(* CODESYS project TASK3.project
   CompiledLibraryCompatibilityVersion: LeadSysStudio V3.5 SP15 Patch 4
   Title: TASK3

Project tree, tasks and I/O mapping:
  Device : PMC600, Leadshine Technology Co., Ltd., order no. 600101, version 3.5.15.40
    application Application
      libraries: Standard, * (System)
      task MainTask (cyclic, interval t#4ms, priority 4, watchdog t#5000ms x 1) calls nothing
      task EtherCAT_Master_Leadshine_A (cyclic, interval 4000 µs, priority 0) calls PLC_PRG, EtherCAT_Master_Leadshine_A.EtherCAT_Task
      task SoftMotion_PlanningTask (freewheeling, priority 15) calls nothing
      program PLC_PRG [LD]
      axis group Tripod: TRAFO.Kin_Tripod_Rotary, axes Axis_3, Axis_4, Axis_5
    Device Diagnose
    Network Configuration
      LocalBus Config
    Resource Usage
    SoftMotion General Axis Pool
    High_Speed_IO_Module : High Speed IO Module, Leadshine Technology Co., Ltd., version 3.5.15.40
        unmapped channels: Genral_IO_IN, Genral_IO_Out
    EtherCAT_Master_Leadshine_A : EtherCAT Master Leadshine, Leadshine Technology Co., Ltd., version 3.5.9.50
        settings: MasterCycleTime = 4000
      PM32EC_LOCAL : PM32EC-LOCAL, Leadshine Technology Co., Ltd., order no. PM32EC-LOCAL, version Revision=16#20061010
          settings: StationAlias = 0; DC sync0 cycletime = 4000; DC sync1 cycletime = 4000
      DM3C_EC522 : DM3C-EC522(COE), Leadshine Technology Co.,Ltd., order no. DM3C-EC522, version Revision=16#00000001
          settings: StationAlias = 0; DC sync0 cycletime = 4000; DC sync1 cycletime = 4000; Number of SDO = 6; Homing method.Index = 16#6098; Homing method.Subindex = 16#00; Homing method.Value = 29; Homing method.Size = 8; Homing method.AbortIfError = FALSE; Homing method.JumpToLine = FALSE; Homing method.Line = 0; Homing method.CompleteAccess = FALSE; Homing velocity (fast).Index = 16#6099; Homing velocity (fast).Subindex = 16#01; Homing velocity (fast).Value = 1667; Homing velocity (fast).Size = 32; Homing velocity (fast).AbortIfError = FALSE; Homing velocity (fast).JumpToLine = FALSE; Homing velocity (fast).Line = 0; Homing velocity (fast).CompleteAccess = FALSE; Homing velocity (slow).Index = 16#6099; Homing velocity (slow).Subindex = 16#02; Homing velocity (slow).Value = 333; Homing velocity (slow).Size = 32; Homing velocity (slow).AbortIfError = FALSE; Homing velocity (slow).JumpToLine = FALSE; Homing velocity (slow).Line = 0; Homing velocity (slow).CompleteAccess = FALSE; Homing acceleration.Index = 16#609A; Homing acceleration.Subindex = 16#00; Homing acceleration.Value = 16667; Homing acceleration.Size = 32; Homing acceleration.AbortIfError = FALSE; Homing acceleration.JumpToLine = FALSE; Homing acceleration.Line = 0; Homing acceleration.CompleteAccess = FALSE; Homing offset.Index = 16#607C; Homing offset.Subindex = 16#00; Homing offset.Value = 0; Homing offset.Size = 32;
            Homing offset.AbortIfError = FALSE; Homing offset.JumpToLine = FALSE; Homing offset.Line = 0; Homing offset.CompleteAccess = FALSE
          unmapped channels: Control Word, Profile Target Position, Touch Probe Function, Last Error Code, Status Word, Modes of Operation display, Position Actual Value, Touch Probe Status, Touch Probe 1 Positive Value, Digital Inputs
        Axis : Axis, 3S - Smart Software Solutions GmbH, order no. 0, version 4.6.1.0
            settings: wDriveID = 0; dwRatioTechUnitsDenom = 500; iRatioTechUnitsNum = 3; 一圈脉冲数 = 10000; 工作台一圈的位移 = 60; 电子齿轮比分子 = 1; 电子齿轮比分母 = 1; ScalingIncs = 500; ScalingUnits = 3; AdrOffset_8010 = 4; BitOffset_8010 = 0; BitLength_8010 = 16; Address_8010 = '%QW2'; Type_8010 = 'UINT'; AddressPointer_8010 = ADR(%QW2); AdrOffset_8020 = 8; BitOffset_8020 = 0; BitLength_8020 = 32; Address_8020 = '%QD2'; Type_8020 = 'DINT'; AddressPointer_8020 = ADR(%QD2); AdrOffset_8030 = 4294967295; BitOffset_8030 = 0; BitLength_8030 = 32; Address_8030 = ''; Type_8030 = 'DINT'; AddressPointer_8030 = 0; AdrOffset_8040 = 4294967295; BitOffset_8040 = 0; BitLength_8040 = 0; Address_8040 = ''; Type_8040 = ''; AddressPointer_8040 = 0; AdrOffset_8050 = 4294967295; BitOffset_8050 = 0; BitLength_8050 = 8; Address_8050 = ''; Type_8050 = 'USINT'; AddressPointer_8050 = 0; AdrOffset_8060 = 12;
              BitOffset_8060 = 0; BitLength_8060 = 16; Address_8060 = '%QW6'; Type_8060 = 'UINT'; AddressPointer_8060 = ADR(%QW6); AdrOffset_8070 = 4294967295; BitOffset_8070 = 0; BitLength_8070 = 0; Address_8070 = ''; Type_8070 = ''; AddressPointer_8070 = 0; AdrOffset_8080 = 4294967295; BitOffset_8080 = 0; BitLength_8080 = 0; Address_8080 = ''; Type_8080 = ''; AddressPointer_8080 = 0; AdrOffset_8090 = 4294967295; BitOffset_8090 = 0; BitLength_8090 = 0; Address_8090 = ''; Type_8090 = ''; AddressPointer_8090 = 0; AdrOffset_8510 = 6; BitOffset_8510 = 0; BitLength_8510 = 16; Address_8510 = '%IW3'; Type_8510 = 'UINT'; AddressPointer_8510 = ADR(%IW3); AdrOffset_8520 = 12; BitOffset_8520 = 0; BitLength_8520 = 32; Address_8520 = '%ID3'; Type_8520 = 'DINT'; AddressPointer_8520 = ADR(%ID3); AdrOffset_8530 = 4294967295; BitOffset_8530 = 0; BitLength_8530 = 0; Address_8530 = ''; Type_8530 = '';
              AddressPointer_8530 = 0; AdrOffset_8540 = 4294967295; BitOffset_8540 = 0; BitLength_8540 = 0; Address_8540 = ''; Type_8540 = ''; AddressPointer_8540 = 0; AdrOffset_8550 = 8; BitOffset_8550 = 0; BitLength_8550 = 8; Address_8550 = '%IB8'; Type_8550 = 'SINT'; AddressPointer_8550 = ADR(%IB8); AdrOffset_8560 = 24; BitOffset_8560 = 0; BitLength_8560 = 32; Address_8560 = '%ID6'; Type_8560 = 'UDINT'; AddressPointer_8560 = ADR(%ID6); AdrOffset_8570 = 16; BitOffset_8570 = 0; BitLength_8570 = 16; Address_8570 = '%IW8'; Type_8570 = 'UINT'; AddressPointer_8570 = ADR(%IW8); AdrOffset_8580 = 20; BitOffset_8580 = 0; BitLength_8580 = 32; Address_8580 = '%ID5'; Type_8580 = 'DINT'; AddressPointer_8580 = ADR(%ID5); AdrOffset_8590 = 4294967295; BitOffset_8590 = 0; BitLength_8590 = 0; Address_8590 = ''; Type_8590 = ''; AddressPointer_8590 = 0; AdrOffset_8600 = 4294967295; BitOffset_8600 = 0; BitLength_8600 = 0;
              Address_8600 = ''; Type_8600 = ''; AddressPointer_8600 = 0; AdrOffset_8600 = 4294967295; BitOffset_8600 = 0; BitLength_8600 = 0; Address_8610 = ''; Type_8610 = ''; AddressPointer_8610 = 0; AdrOffset_8620 = 4294967295; BitOffset_8620 = 0; BitLength_8620 = 0; Address_8620 = ''; Type_8620 = ''; AddressPointer_8620 = 0
      DM3C_EC522_1 : DM3C-EC522(COE), Leadshine Technology Co.,Ltd., order no. DM3C-EC522, version Revision=16#00000001
          settings: StationAlias = 0; DC sync0 cycletime = 4000; DC sync1 cycletime = 4000; Number of SDO = 6; Homing method.Index = 16#6098; Homing method.Subindex = 16#00; Homing method.Value = 29; Homing method.Size = 8; Homing method.AbortIfError = FALSE; Homing method.JumpToLine = FALSE; Homing method.Line = 0; Homing method.CompleteAccess = FALSE; Homing velocity (fast).Index = 16#6099; Homing velocity (fast).Subindex = 16#01; Homing velocity (fast).Value = 1667; Homing velocity (fast).Size = 32; Homing velocity (fast).AbortIfError = FALSE; Homing velocity (fast).JumpToLine = FALSE; Homing velocity (fast).Line = 0; Homing velocity (fast).CompleteAccess = FALSE; Homing velocity (slow).Index = 16#6099; Homing velocity (slow).Subindex = 16#02; Homing velocity (slow).Value = 333; Homing velocity (slow).Size = 32; Homing velocity (slow).AbortIfError = FALSE; Homing velocity (slow).JumpToLine = FALSE; Homing velocity (slow).Line = 0; Homing velocity (slow).CompleteAccess = FALSE; Homing acceleration.Index = 16#609A; Homing acceleration.Subindex = 16#00; Homing acceleration.Value = 16667; Homing acceleration.Size = 32; Homing acceleration.AbortIfError = FALSE; Homing acceleration.JumpToLine = FALSE; Homing acceleration.Line = 0; Homing acceleration.CompleteAccess = FALSE; Homing offset.Index = 16#607C; Homing offset.Subindex = 16#00; Homing offset.Value = 0; Homing offset.Size = 32;
            Homing offset.AbortIfError = FALSE; Homing offset.JumpToLine = FALSE; Homing offset.Line = 0; Homing offset.CompleteAccess = FALSE
          unmapped channels: Control Word, Profile Target Position, Touch Probe Function, Last Error Code, Status Word, Modes of Operation display, Position Actual Value, Touch Probe Status, Touch Probe 1 Positive Value, Digital Inputs
        Axis_1 : Axis, 3S - Smart Software Solutions GmbH, order no. 0, version 4.6.1.0
            settings: dwRatioTechUnitsDenom = 500; iRatioTechUnitsNum = 3; 一圈脉冲数 = 10000; 工作台一圈的位移 = 60; 电子齿轮比分子 = 1; 电子齿轮比分母 = 1; ScalingIncs = 500; ScalingUnits = 3; AdrOffset_8010 = 16; BitOffset_8010 = 0; BitLength_8010 = 16; Address_8010 = '%QW8'; Type_8010 = 'UINT'; AddressPointer_8010 = ADR(%QW8); AdrOffset_8020 = 20; BitOffset_8020 = 0; BitLength_8020 = 32; Address_8020 = '%QD5'; Type_8020 = 'DINT'; AddressPointer_8020 = ADR(%QD5); AdrOffset_8030 = 4294967295; BitOffset_8030 = 0; BitLength_8030 = 32; Address_8030 = ''; Type_8030 = 'DINT'; AddressPointer_8030 = 0; AdrOffset_8040 = 4294967295; BitOffset_8040 = 0; BitLength_8040 = 0; Address_8040 = ''; Type_8040 = ''; AddressPointer_8040 = 0; AdrOffset_8050 = 4294967295; BitOffset_8050 = 0; BitLength_8050 = 8; Address_8050 = ''; Type_8050 = 'USINT'; AddressPointer_8050 = 0; AdrOffset_8060 = 24; BitOffset_8060 = 0;
              BitLength_8060 = 16; Address_8060 = '%QW12'; Type_8060 = 'UINT'; AddressPointer_8060 = ADR(%QW12); AdrOffset_8070 = 4294967295; BitOffset_8070 = 0; BitLength_8070 = 0; Address_8070 = ''; Type_8070 = ''; AddressPointer_8070 = 0; AdrOffset_8080 = 4294967295; BitOffset_8080 = 0; BitLength_8080 = 0; Address_8080 = ''; Type_8080 = ''; AddressPointer_8080 = 0; AdrOffset_8090 = 4294967295; BitOffset_8090 = 0; BitLength_8090 = 0; Address_8090 = ''; Type_8090 = ''; AddressPointer_8090 = 0; AdrOffset_8510 = 30; BitOffset_8510 = 0; BitLength_8510 = 16; Address_8510 = '%IW15'; Type_8510 = 'UINT'; AddressPointer_8510 = ADR(%IW15); AdrOffset_8520 = 36; BitOffset_8520 = 0; BitLength_8520 = 32; Address_8520 = '%ID9'; Type_8520 = 'DINT'; AddressPointer_8520 = ADR(%ID9); AdrOffset_8530 = 4294967295; BitOffset_8530 = 0; BitLength_8530 = 0; Address_8530 = ''; Type_8530 = ''; AddressPointer_8530 = 0;
              AdrOffset_8540 = 4294967295; BitOffset_8540 = 0; BitLength_8540 = 0; Address_8540 = ''; Type_8540 = ''; AddressPointer_8540 = 0; AdrOffset_8550 = 32; BitOffset_8550 = 0; BitLength_8550 = 8; Address_8550 = '%IB32'; Type_8550 = 'SINT'; AddressPointer_8550 = ADR(%IB32); AdrOffset_8560 = 48; BitOffset_8560 = 0; BitLength_8560 = 32; Address_8560 = '%ID12'; Type_8560 = 'UDINT'; AddressPointer_8560 = ADR(%ID12); AdrOffset_8570 = 40; BitOffset_8570 = 0; BitLength_8570 = 16; Address_8570 = '%IW20'; Type_8570 = 'UINT'; AddressPointer_8570 = ADR(%IW20); AdrOffset_8580 = 44; BitOffset_8580 = 0; BitLength_8580 = 32; Address_8580 = '%ID11'; Type_8580 = 'DINT'; AddressPointer_8580 = ADR(%ID11); AdrOffset_8590 = 4294967295; BitOffset_8590 = 0; BitLength_8590 = 0; Address_8590 = ''; Type_8590 = ''; AddressPointer_8590 = 0; AdrOffset_8600 = 4294967295; BitOffset_8600 = 0; BitLength_8600 = 0; Address_8600 = '';
              Type_8600 = ''; AddressPointer_8600 = 0; AdrOffset_8600 = 4294967295; BitOffset_8600 = 0; BitLength_8600 = 0; Address_8610 = ''; Type_8610 = ''; AddressPointer_8610 = 0; AdrOffset_8620 = 4294967295; BitOffset_8620 = 0; BitLength_8620 = 0; Address_8620 = ''; Type_8620 = ''; AddressPointer_8620 = 0
      DM3C_EC522_2 : DM3C-EC522(COE), Leadshine Technology Co.,Ltd., order no. DM3C-EC522, version Revision=16#00000001
          settings: StationAlias = 0; DC sync0 cycletime = 4000; DC sync1 cycletime = 4000; Number of SDO = 6; Homing method.Index = 16#6098; Homing method.Subindex = 16#00; Homing method.Value = 29; Homing method.Size = 8; Homing method.AbortIfError = FALSE; Homing method.JumpToLine = FALSE; Homing method.Line = 0; Homing method.CompleteAccess = FALSE; Homing velocity (fast).Index = 16#6099; Homing velocity (fast).Subindex = 16#01; Homing velocity (fast).Value = 25000; Homing velocity (fast).Size = 32; Homing velocity (fast).AbortIfError = FALSE; Homing velocity (fast).JumpToLine = FALSE; Homing velocity (fast).Line = 0; Homing velocity (fast).CompleteAccess = FALSE; Homing velocity (slow).Index = 16#6099; Homing velocity (slow).Subindex = 16#02; Homing velocity (slow).Value = 5000; Homing velocity (slow).Size = 32; Homing velocity (slow).AbortIfError = FALSE; Homing velocity (slow).JumpToLine = FALSE; Homing velocity (slow).Line = 0; Homing velocity (slow).CompleteAccess = FALSE; Homing acceleration.Index = 16#609A; Homing acceleration.Subindex = 16#00; Homing acceleration.Value = 250000; Homing acceleration.Size = 32; Homing acceleration.AbortIfError = FALSE; Homing acceleration.JumpToLine = FALSE; Homing acceleration.Line = 0; Homing acceleration.CompleteAccess = FALSE; Homing offset.Index = 16#607C; Homing offset.Subindex = 16#00; Homing offset.Value = 0; Homing offset.Size = 32;
            Homing offset.AbortIfError = FALSE; Homing offset.JumpToLine = FALSE; Homing offset.Line = 0; Homing offset.CompleteAccess = FALSE
          unmapped channels: Control Word, Profile Target Position, Touch Probe Function, Last Error Code, Status Word, Modes of Operation display, Position Actual Value, Touch Probe Status, Touch Probe 1 Positive Value, Digital Inputs
        Axis_2 : Axis, 3S - Smart Software Solutions GmbH, order no. 0, version 4.6.1.0
            settings: wDriveID = 2; dwRatioTechUnitsDenom = 2500; 一圈脉冲数 = 10000; 工作台一圈的位移 = 4; 电子齿轮比分子 = 1; 电子齿轮比分母 = 1; ScalingIncs = 2500; AdrOffset_8010 = 28; BitOffset_8010 = 0; BitLength_8010 = 16; Address_8010 = '%QW14'; Type_8010 = 'UINT'; AddressPointer_8010 = ADR(%QW14); AdrOffset_8020 = 32; BitOffset_8020 = 0; BitLength_8020 = 32; Address_8020 = '%QD8'; Type_8020 = 'DINT'; AddressPointer_8020 = ADR(%QD8); AdrOffset_8030 = 4294967295; BitOffset_8030 = 0; BitLength_8030 = 32; Address_8030 = ''; Type_8030 = 'DINT'; AddressPointer_8030 = 0; AdrOffset_8040 = 4294967295; BitOffset_8040 = 0; BitLength_8040 = 0; Address_8040 = ''; Type_8040 = ''; AddressPointer_8040 = 0; AdrOffset_8050 = 4294967295; BitOffset_8050 = 0; BitLength_8050 = 8; Address_8050 = ''; Type_8050 = 'USINT'; AddressPointer_8050 = 0; AdrOffset_8060 = 36; BitOffset_8060 = 0; BitLength_8060 = 16;
              Address_8060 = '%QW18'; Type_8060 = 'UINT'; AddressPointer_8060 = ADR(%QW18); AdrOffset_8070 = 4294967295; BitOffset_8070 = 0; BitLength_8070 = 0; Address_8070 = ''; Type_8070 = ''; AddressPointer_8070 = 0; AdrOffset_8080 = 4294967295; BitOffset_8080 = 0; BitLength_8080 = 0; Address_8080 = ''; Type_8080 = ''; AddressPointer_8080 = 0; AdrOffset_8090 = 4294967295; BitOffset_8090 = 0; BitLength_8090 = 0; Address_8090 = ''; Type_8090 = ''; AddressPointer_8090 = 0; AdrOffset_8510 = 54; BitOffset_8510 = 0; BitLength_8510 = 16; Address_8510 = '%IW27'; Type_8510 = 'UINT'; AddressPointer_8510 = ADR(%IW27); AdrOffset_8520 = 60; BitOffset_8520 = 0; BitLength_8520 = 32; Address_8520 = '%ID15'; Type_8520 = 'DINT'; AddressPointer_8520 = ADR(%ID15); AdrOffset_8530 = 4294967295; BitOffset_8530 = 0; BitLength_8530 = 0; Address_8530 = ''; Type_8530 = ''; AddressPointer_8530 = 0; AdrOffset_8540 = 4294967295;
              BitOffset_8540 = 0; BitLength_8540 = 0; Address_8540 = ''; Type_8540 = ''; AddressPointer_8540 = 0; AdrOffset_8550 = 56; BitOffset_8550 = 0; BitLength_8550 = 8; Address_8550 = '%IB56'; Type_8550 = 'SINT'; AddressPointer_8550 = ADR(%IB56); AdrOffset_8560 = 72; BitOffset_8560 = 0; BitLength_8560 = 32; Address_8560 = '%ID18'; Type_8560 = 'UDINT'; AddressPointer_8560 = ADR(%ID18); AdrOffset_8570 = 64; BitOffset_8570 = 0; BitLength_8570 = 16; Address_8570 = '%IW32'; Type_8570 = 'UINT'; AddressPointer_8570 = ADR(%IW32); AdrOffset_8580 = 68; BitOffset_8580 = 0; BitLength_8580 = 32; Address_8580 = '%ID17'; Type_8580 = 'DINT'; AddressPointer_8580 = ADR(%ID17); AdrOffset_8590 = 4294967295; BitOffset_8590 = 0; BitLength_8590 = 0; Address_8590 = ''; Type_8590 = ''; AddressPointer_8590 = 0; AdrOffset_8600 = 4294967295; BitOffset_8600 = 0; BitLength_8600 = 0; Address_8600 = ''; Type_8600 = '';
              AddressPointer_8600 = 0; AdrOffset_8600 = 4294967295; BitOffset_8600 = 0; BitLength_8600 = 0; Address_8610 = ''; Type_8610 = ''; AddressPointer_8610 = 0; AdrOffset_8620 = 4294967295; BitOffset_8620 = 0; BitLength_8620 = 0; Address_8620 = ''; Type_8620 = ''; AddressPointer_8620 = 0
      DM3C_EC522_3 : DM3C-EC522(COE), Leadshine Technology Co.,Ltd., order no. DM3C-EC522, version Revision=16#00000001
          settings: StationAlias = 0; DC sync0 cycletime = 4000; DC sync1 cycletime = 4000; Number of SDO = 6; Homing method.Index = 16#6098; Homing method.Subindex = 16#00; Homing method.Value = 21; Homing method.Size = 8; Homing method.AbortIfError = FALSE; Homing method.JumpToLine = FALSE; Homing method.Line = 0; Homing method.CompleteAccess = FALSE; Homing velocity (fast).Index = 16#6099; Homing velocity (fast).Subindex = 16#01; Homing velocity (fast).Value = 7500; Homing velocity (fast).Size = 32; Homing velocity (fast).AbortIfError = FALSE; Homing velocity (fast).JumpToLine = FALSE; Homing velocity (fast).Line = 0; Homing velocity (fast).CompleteAccess = FALSE; Homing velocity (slow).Index = 16#6099; Homing velocity (slow).Subindex = 16#02; Homing velocity (slow).Value = 5000; Homing velocity (slow).Size = 32; Homing velocity (slow).AbortIfError = FALSE; Homing velocity (slow).JumpToLine = FALSE; Homing velocity (slow).Line = 0; Homing velocity (slow).CompleteAccess = FALSE; Homing acceleration.Index = 16#609A; Homing acceleration.Subindex = 16#00; Homing acceleration.Value = 50000; Homing acceleration.Size = 32; Homing acceleration.AbortIfError = FALSE; Homing acceleration.JumpToLine = FALSE; Homing acceleration.Line = 0; Homing acceleration.CompleteAccess = FALSE; Homing offset.Index = 16#607C; Homing offset.Subindex = 16#00; Homing offset.Value = 0; Homing offset.Size = 32;
            Homing offset.AbortIfError = FALSE; Homing offset.JumpToLine = FALSE; Homing offset.Line = 0; Homing offset.CompleteAccess = FALSE
          unmapped channels: Control Word, Profile Target Position, Touch Probe Function, Last Error Code, Status Word, Modes of Operation display, Position Actual Value, Touch Probe Status, Touch Probe 1 Positive Value, Digital Inputs
        Axis_3 : Axis, 3S - Smart Software Solutions GmbH, order no. 0, version 4.6.1.0
            settings: wDriveID = 3; dwRatioTechUnitsDenom = 500; iRatioTechUnitsNum = -1; 一圈脉冲数 = 36000; 工作台一圈的位移 = 360; 电子齿轮比分子 = 5; 电子齿轮比分母 = 1; ScalingIncs = 500; InvertDirection = True; AdrOffset_8010 = 40; BitOffset_8010 = 0; BitLength_8010 = 16; Address_8010 = '%QW20'; Type_8010 = 'UINT'; AddressPointer_8010 = ADR(%QW20); AdrOffset_8020 = 44; BitOffset_8020 = 0; BitLength_8020 = 32; Address_8020 = '%QD11'; Type_8020 = 'DINT'; AddressPointer_8020 = ADR(%QD11); AdrOffset_8030 = 4294967295; BitOffset_8030 = 0; BitLength_8030 = 32; Address_8030 = ''; Type_8030 = 'DINT'; AddressPointer_8030 = 0; AdrOffset_8040 = 4294967295; BitOffset_8040 = 0; BitLength_8040 = 0; Address_8040 = ''; Type_8040 = ''; AddressPointer_8040 = 0; AdrOffset_8050 = 4294967295; BitOffset_8050 = 0; BitLength_8050 = 8; Address_8050 = ''; Type_8050 = 'USINT'; AddressPointer_8050 = 0; AdrOffset_8060 = 48;
              BitOffset_8060 = 0; BitLength_8060 = 16; Address_8060 = '%QW24'; Type_8060 = 'UINT'; AddressPointer_8060 = ADR(%QW24); AdrOffset_8070 = 4294967295; BitOffset_8070 = 0; BitLength_8070 = 0; Address_8070 = ''; Type_8070 = ''; AddressPointer_8070 = 0; AdrOffset_8080 = 4294967295; BitOffset_8080 = 0; BitLength_8080 = 0; Address_8080 = ''; Type_8080 = ''; AddressPointer_8080 = 0; AdrOffset_8090 = 4294967295; BitOffset_8090 = 0; BitLength_8090 = 0; Address_8090 = ''; Type_8090 = ''; AddressPointer_8090 = 0; AdrOffset_8510 = 78; BitOffset_8510 = 0; BitLength_8510 = 16; Address_8510 = '%IW39'; Type_8510 = 'UINT'; AddressPointer_8510 = ADR(%IW39); AdrOffset_8520 = 84; BitOffset_8520 = 0; BitLength_8520 = 32; Address_8520 = '%ID21'; Type_8520 = 'DINT'; AddressPointer_8520 = ADR(%ID21); AdrOffset_8530 = 4294967295; BitOffset_8530 = 0; BitLength_8530 = 0; Address_8530 = ''; Type_8530 = '';
              AddressPointer_8530 = 0; AdrOffset_8540 = 4294967295; BitOffset_8540 = 0; BitLength_8540 = 0; Address_8540 = ''; Type_8540 = ''; AddressPointer_8540 = 0; AdrOffset_8550 = 80; BitOffset_8550 = 0; BitLength_8550 = 8; Address_8550 = '%IB80'; Type_8550 = 'SINT'; AddressPointer_8550 = ADR(%IB80); AdrOffset_8560 = 96; BitOffset_8560 = 0; BitLength_8560 = 32; Address_8560 = '%ID24'; Type_8560 = 'UDINT'; AddressPointer_8560 = ADR(%ID24); AdrOffset_8570 = 88; BitOffset_8570 = 0; BitLength_8570 = 16; Address_8570 = '%IW44'; Type_8570 = 'UINT'; AddressPointer_8570 = ADR(%IW44); AdrOffset_8580 = 92; BitOffset_8580 = 0; BitLength_8580 = 32; Address_8580 = '%ID23'; Type_8580 = 'DINT'; AddressPointer_8580 = ADR(%ID23); AdrOffset_8590 = 4294967295; BitOffset_8590 = 0; BitLength_8590 = 0; Address_8590 = ''; Type_8590 = ''; AddressPointer_8590 = 0; AdrOffset_8600 = 4294967295; BitOffset_8600 = 0; BitLength_8600 = 0;
              Address_8600 = ''; Type_8600 = ''; AddressPointer_8600 = 0; AdrOffset_8600 = 4294967295; BitOffset_8600 = 0; BitLength_8600 = 0; Address_8610 = ''; Type_8610 = ''; AddressPointer_8610 = 0; AdrOffset_8620 = 4294967295; BitOffset_8620 = 0; BitLength_8620 = 0; Address_8620 = ''; Type_8620 = ''; AddressPointer_8620 = 0
      DM3C_EC522_4 : DM3C-EC522(COE), Leadshine Technology Co.,Ltd., order no. DM3C-EC522, version Revision=16#00000001
          settings: StationAlias = 0; DC sync0 cycletime = 4000; DC sync1 cycletime = 4000; Number of SDO = 6; Homing method.Index = 16#6098; Homing method.Subindex = 16#00; Homing method.Value = 21; Homing method.Size = 8; Homing method.AbortIfError = FALSE; Homing method.JumpToLine = FALSE; Homing method.Line = 0; Homing method.CompleteAccess = FALSE; Homing velocity (fast).Index = 16#6099; Homing velocity (fast).Subindex = 16#01; Homing velocity (fast).Value = 7500; Homing velocity (fast).Size = 32; Homing velocity (fast).AbortIfError = FALSE; Homing velocity (fast).JumpToLine = FALSE; Homing velocity (fast).Line = 0; Homing velocity (fast).CompleteAccess = FALSE; Homing velocity (slow).Index = 16#6099; Homing velocity (slow).Subindex = 16#02; Homing velocity (slow).Value = 5000; Homing velocity (slow).Size = 32; Homing velocity (slow).AbortIfError = FALSE; Homing velocity (slow).JumpToLine = FALSE; Homing velocity (slow).Line = 0; Homing velocity (slow).CompleteAccess = FALSE; Homing acceleration.Index = 16#609A; Homing acceleration.Subindex = 16#00; Homing acceleration.Value = 50000; Homing acceleration.Size = 32; Homing acceleration.AbortIfError = FALSE; Homing acceleration.JumpToLine = FALSE; Homing acceleration.Line = 0; Homing acceleration.CompleteAccess = FALSE; Homing offset.Index = 16#607C; Homing offset.Subindex = 16#00; Homing offset.Value = 0; Homing offset.Size = 32;
            Homing offset.AbortIfError = FALSE; Homing offset.JumpToLine = FALSE; Homing offset.Line = 0; Homing offset.CompleteAccess = FALSE
          unmapped channels: Control Word, Profile Target Position, Touch Probe Function, Last Error Code, Status Word, Modes of Operation display, Position Actual Value, Touch Probe Status, Touch Probe 1 Positive Value, Digital Inputs
        Axis_4 : Axis, 3S - Smart Software Solutions GmbH, order no. 0, version 4.6.1.0
            settings: wDriveID = 4; dwRatioTechUnitsDenom = 500; iRatioTechUnitsNum = -1; 一圈脉冲数 = 36000; 工作台一圈的位移 = 360; 电子齿轮比分子 = 5; 电子齿轮比分母 = 1; ScalingIncs = 500; InvertDirection = True; AdrOffset_8010 = 52; BitOffset_8010 = 0; BitLength_8010 = 16; Address_8010 = '%QW26'; Type_8010 = 'UINT'; AddressPointer_8010 = ADR(%QW26); AdrOffset_8020 = 56; BitOffset_8020 = 0; BitLength_8020 = 32; Address_8020 = '%QD14'; Type_8020 = 'DINT'; AddressPointer_8020 = ADR(%QD14); AdrOffset_8030 = 4294967295; BitOffset_8030 = 0; BitLength_8030 = 32; Address_8030 = ''; Type_8030 = 'DINT'; AddressPointer_8030 = 0; AdrOffset_8040 = 4294967295; BitOffset_8040 = 0; BitLength_8040 = 0; Address_8040 = ''; Type_8040 = ''; AddressPointer_8040 = 0; AdrOffset_8050 = 4294967295; BitOffset_8050 = 0; BitLength_8050 = 8; Address_8050 = ''; Type_8050 = 'USINT'; AddressPointer_8050 = 0; AdrOffset_8060 = 60;
              BitOffset_8060 = 0; BitLength_8060 = 16; Address_8060 = '%QW30'; Type_8060 = 'UINT'; AddressPointer_8060 = ADR(%QW30); AdrOffset_8070 = 4294967295; BitOffset_8070 = 0; BitLength_8070 = 0; Address_8070 = ''; Type_8070 = ''; AddressPointer_8070 = 0; AdrOffset_8080 = 4294967295; BitOffset_8080 = 0; BitLength_8080 = 0; Address_8080 = ''; Type_8080 = ''; AddressPointer_8080 = 0; AdrOffset_8090 = 4294967295; BitOffset_8090 = 0; BitLength_8090 = 0; Address_8090 = ''; Type_8090 = ''; AddressPointer_8090 = 0; AdrOffset_8510 = 102; BitOffset_8510 = 0; BitLength_8510 = 16; Address_8510 = '%IW51'; Type_8510 = 'UINT'; AddressPointer_8510 = ADR(%IW51); AdrOffset_8520 = 108; BitOffset_8520 = 0; BitLength_8520 = 32; Address_8520 = '%ID27'; Type_8520 = 'DINT'; AddressPointer_8520 = ADR(%ID27); AdrOffset_8530 = 4294967295; BitOffset_8530 = 0; BitLength_8530 = 0; Address_8530 = ''; Type_8530 = '';
              AddressPointer_8530 = 0; AdrOffset_8540 = 4294967295; BitOffset_8540 = 0; BitLength_8540 = 0; Address_8540 = ''; Type_8540 = ''; AddressPointer_8540 = 0; AdrOffset_8550 = 104; BitOffset_8550 = 0; BitLength_8550 = 8; Address_8550 = '%IB104'; Type_8550 = 'SINT'; AddressPointer_8550 = ADR(%IB104); AdrOffset_8560 = 120; BitOffset_8560 = 0; BitLength_8560 = 32; Address_8560 = '%ID30'; Type_8560 = 'UDINT'; AddressPointer_8560 = ADR(%ID30); AdrOffset_8570 = 112; BitOffset_8570 = 0; BitLength_8570 = 16; Address_8570 = '%IW56'; Type_8570 = 'UINT'; AddressPointer_8570 = ADR(%IW56); AdrOffset_8580 = 116; BitOffset_8580 = 0; BitLength_8580 = 32; Address_8580 = '%ID29'; Type_8580 = 'DINT'; AddressPointer_8580 = ADR(%ID29); AdrOffset_8590 = 4294967295; BitOffset_8590 = 0; BitLength_8590 = 0; Address_8590 = ''; Type_8590 = ''; AddressPointer_8590 = 0; AdrOffset_8600 = 4294967295; BitOffset_8600 = 0; BitLength_8600 = 0;
              Address_8600 = ''; Type_8600 = ''; AddressPointer_8600 = 0; AdrOffset_8600 = 4294967295; BitOffset_8600 = 0; BitLength_8600 = 0; Address_8610 = ''; Type_8610 = ''; AddressPointer_8610 = 0; AdrOffset_8620 = 4294967295; BitOffset_8620 = 0; BitLength_8620 = 0; Address_8620 = ''; Type_8620 = ''; AddressPointer_8620 = 0
      DM3C_EC522_5 : DM3C-EC522(COE), Leadshine Technology Co.,Ltd., order no. DM3C-EC522, version Revision=16#00000001
          settings: StationAlias = 0; DC sync0 cycletime = 4000; DC sync1 cycletime = 4000; Number of SDO = 6; Homing method.Index = 16#6098; Homing method.Subindex = 16#00; Homing method.Value = 21; Homing method.Size = 8; Homing method.AbortIfError = FALSE; Homing method.JumpToLine = FALSE; Homing method.Line = 0; Homing method.CompleteAccess = FALSE; Homing velocity (fast).Index = 16#6099; Homing velocity (fast).Subindex = 16#01; Homing velocity (fast).Value = 7500; Homing velocity (fast).Size = 32; Homing velocity (fast).AbortIfError = FALSE; Homing velocity (fast).JumpToLine = FALSE; Homing velocity (fast).Line = 0; Homing velocity (fast).CompleteAccess = FALSE; Homing velocity (slow).Index = 16#6099; Homing velocity (slow).Subindex = 16#02; Homing velocity (slow).Value = 5000; Homing velocity (slow).Size = 32; Homing velocity (slow).AbortIfError = FALSE; Homing velocity (slow).JumpToLine = FALSE; Homing velocity (slow).Line = 0; Homing velocity (slow).CompleteAccess = FALSE; Homing acceleration.Index = 16#609A; Homing acceleration.Subindex = 16#00; Homing acceleration.Value = 50000; Homing acceleration.Size = 32; Homing acceleration.AbortIfError = FALSE; Homing acceleration.JumpToLine = FALSE; Homing acceleration.Line = 0; Homing acceleration.CompleteAccess = FALSE; Homing offset.Index = 16#607C; Homing offset.Subindex = 16#00; Homing offset.Value = 0; Homing offset.Size = 32;
            Homing offset.AbortIfError = FALSE; Homing offset.JumpToLine = FALSE; Homing offset.Line = 0; Homing offset.CompleteAccess = FALSE
          unmapped channels: Control Word, Profile Target Position, Touch Probe Function, Last Error Code, Status Word, Modes of Operation display, Position Actual Value, Touch Probe Status, Touch Probe 1 Positive Value, Digital Inputs
        Axis_5 : Axis, 3S - Smart Software Solutions GmbH, order no. 0, version 4.6.1.0
            settings: wDriveID = 5; dwRatioTechUnitsDenom = 500; iRatioTechUnitsNum = -1; 一圈脉冲数 = 36000; 工作台一圈的位移 = 360; 电子齿轮比分子 = 5; 电子齿轮比分母 = 1; ScalingIncs = 500; InvertDirection = True; AdrOffset_8010 = 64; BitOffset_8010 = 0; BitLength_8010 = 16; Address_8010 = '%QW32'; Type_8010 = 'UINT'; AddressPointer_8010 = ADR(%QW32); AdrOffset_8020 = 68; BitOffset_8020 = 0; BitLength_8020 = 32; Address_8020 = '%QD17'; Type_8020 = 'DINT'; AddressPointer_8020 = ADR(%QD17); AdrOffset_8030 = 4294967295; BitOffset_8030 = 0; BitLength_8030 = 32; Address_8030 = ''; Type_8030 = 'DINT'; AddressPointer_8030 = 0; AdrOffset_8040 = 4294967295; BitOffset_8040 = 0; BitLength_8040 = 0; Address_8040 = ''; Type_8040 = ''; AddressPointer_8040 = 0; AdrOffset_8050 = 4294967295; BitOffset_8050 = 0; BitLength_8050 = 8; Address_8050 = ''; Type_8050 = 'USINT'; AddressPointer_8050 = 0; AdrOffset_8060 = 72;
              BitOffset_8060 = 0; BitLength_8060 = 16; Address_8060 = '%QW36'; Type_8060 = 'UINT'; AddressPointer_8060 = ADR(%QW36); AdrOffset_8070 = 4294967295; BitOffset_8070 = 0; BitLength_8070 = 0; Address_8070 = ''; Type_8070 = ''; AddressPointer_8070 = 0; AdrOffset_8080 = 4294967295; BitOffset_8080 = 0; BitLength_8080 = 0; Address_8080 = ''; Type_8080 = ''; AddressPointer_8080 = 0; AdrOffset_8090 = 4294967295; BitOffset_8090 = 0; BitLength_8090 = 0; Address_8090 = ''; Type_8090 = ''; AddressPointer_8090 = 0; AdrOffset_8510 = 126; BitOffset_8510 = 0; BitLength_8510 = 16; Address_8510 = '%IW63'; Type_8510 = 'UINT'; AddressPointer_8510 = ADR(%IW63); AdrOffset_8520 = 132; BitOffset_8520 = 0; BitLength_8520 = 32; Address_8520 = '%ID33'; Type_8520 = 'DINT'; AddressPointer_8520 = ADR(%ID33); AdrOffset_8530 = 4294967295; BitOffset_8530 = 0; BitLength_8530 = 0; Address_8530 = ''; Type_8530 = '';
              AddressPointer_8530 = 0; AdrOffset_8540 = 4294967295; BitOffset_8540 = 0; BitLength_8540 = 0; Address_8540 = ''; Type_8540 = ''; AddressPointer_8540 = 0; AdrOffset_8550 = 128; BitOffset_8550 = 0; BitLength_8550 = 8; Address_8550 = '%IB128'; Type_8550 = 'SINT'; AddressPointer_8550 = ADR(%IB128); AdrOffset_8560 = 144; BitOffset_8560 = 0; BitLength_8560 = 32; Address_8560 = '%ID36'; Type_8560 = 'UDINT'; AddressPointer_8560 = ADR(%ID36); AdrOffset_8570 = 136; BitOffset_8570 = 0; BitLength_8570 = 16; Address_8570 = '%IW68'; Type_8570 = 'UINT'; AddressPointer_8570 = ADR(%IW68); AdrOffset_8580 = 140; BitOffset_8580 = 0; BitLength_8580 = 32; Address_8580 = '%ID35'; Type_8580 = 'DINT'; AddressPointer_8580 = ADR(%ID35); AdrOffset_8590 = 4294967295; BitOffset_8590 = 0; BitLength_8590 = 0; Address_8590 = ''; Type_8590 = ''; AddressPointer_8590 = 0; AdrOffset_8600 = 4294967295; BitOffset_8600 = 0; BitLength_8600 = 0;
              Address_8600 = ''; Type_8600 = ''; AddressPointer_8600 = 0; AdrOffset_8600 = 4294967295; BitOffset_8600 = 0; BitLength_8600 = 0; Address_8610 = ''; Type_8610 = ''; AddressPointer_8610 = 0; AdrOffset_8620 = 4294967295; BitOffset_8620 = 0; BitLength_8620 = 0; Address_8620 = ''; Type_8620 = ''; AddressPointer_8620 = 0
      L7EC_100 : L7EC-100(COE), Leadshine Technology Co.,Ltd., order no. L7EC-100, version Revision=16#00000001
          settings: StationAlias = 0; DC sync0 cycletime = 4000; DC sync1 cycletime = 4000; Number of SDO = 6; Homing method.Index = 16#6098; Homing method.Subindex = 16#00; Homing method.Value = 1; Homing method.Size = 8; Homing method.AbortIfError = FALSE; Homing method.JumpToLine = FALSE; Homing method.Line = 0; Homing method.CompleteAccess = FALSE; Homing velocity (fast).Index = 16#6099; Homing velocity (fast).Subindex = 16#01; Homing velocity (fast).Value = 40000; Homing velocity (fast).Size = 32; Homing velocity (fast).AbortIfError = FALSE; Homing velocity (fast).JumpToLine = FALSE; Homing velocity (fast).Line = 0; Homing velocity (fast).CompleteAccess = FALSE; Homing velocity (slow).Index = 16#6099; Homing velocity (slow).Subindex = 16#02; Homing velocity (slow).Value = 8000; Homing velocity (slow).Size = 32; Homing velocity (slow).AbortIfError = FALSE; Homing velocity (slow).JumpToLine = FALSE; Homing velocity (slow).Line = 0; Homing velocity (slow).CompleteAccess = FALSE; Homing acceleration.Index = 16#609A; Homing acceleration.Subindex = 16#00; Homing acceleration.Value = 400000; Homing acceleration.Size = 32; Homing acceleration.AbortIfError = FALSE; Homing acceleration.JumpToLine = FALSE; Homing acceleration.Line = 0; Homing acceleration.CompleteAccess = FALSE; Homing offset.Index = 16#607C; Homing offset.Subindex = 16#00; Homing offset.Value = 0; Homing offset.Size = 32;
            Homing offset.AbortIfError = FALSE; Homing offset.JumpToLine = FALSE; Homing offset.Line = 0; Homing offset.CompleteAccess = FALSE
          unmapped channels: Control word, Profile target position, Touch Probe Function, Last error code, Status word, Modes of operation display, Actual motor position, Touch Probe Status, Touch probe pos1 pos value, Digital inputs
        Axis_6 : Axis, 3S - Smart Software Solutions GmbH, order no. 0, version 4.6.1.0
            settings: wDriveID = 6; dwRatioTechUnitsDenom = 4000; 一圈脉冲数 = 10000; 工作台一圈的位移 = 2.5; 电子齿轮比分子 = 1; 电子齿轮比分母 = 1; ScalingIncs = 4000; AdrOffset_8010 = 76; BitOffset_8010 = 0; BitLength_8010 = 16; Address_8010 = '%QW38'; Type_8010 = 'UINT'; AddressPointer_8010 = ADR(%QW38); AdrOffset_8020 = 80; BitOffset_8020 = 0; BitLength_8020 = 32; Address_8020 = '%QD20'; Type_8020 = 'DINT'; AddressPointer_8020 = ADR(%QD20); AdrOffset_8030 = 4294967295; BitOffset_8030 = 0; BitLength_8030 = 32; Address_8030 = ''; Type_8030 = 'DINT'; AddressPointer_8030 = 0; AdrOffset_8040 = 4294967295; BitOffset_8040 = 0; BitLength_8040 = 16; Address_8040 = ''; Type_8040 = 'INT'; AddressPointer_8040 = 0; AdrOffset_8050 = 4294967295; BitOffset_8050 = 0; BitLength_8050 = 8; Address_8050 = ''; Type_8050 = 'USINT'; AddressPointer_8050 = 0; AdrOffset_8060 = 84; BitOffset_8060 = 0; BitLength_8060 = 16;
              Address_8060 = '%QW42'; Type_8060 = 'UINT'; AddressPointer_8060 = ADR(%QW42); AdrOffset_8070 = 4294967295; BitOffset_8070 = 0; BitLength_8070 = 0; Address_8070 = ''; Type_8070 = ''; AddressPointer_8070 = 0; AdrOffset_8080 = 4294967295; BitOffset_8080 = 0; BitLength_8080 = 16; Address_8080 = ''; Type_8080 = 'INT'; AddressPointer_8080 = 0; AdrOffset_8090 = 4294967295; BitOffset_8090 = 0; BitLength_8090 = 0; Address_8090 = ''; Type_8090 = ''; AddressPointer_8090 = 0; AdrOffset_8510 = 150; BitOffset_8510 = 0; BitLength_8510 = 16; Address_8510 = '%IW75'; Type_8510 = 'UINT'; AddressPointer_8510 = ADR(%IW75); AdrOffset_8520 = 156; BitOffset_8520 = 0; BitLength_8520 = 32; Address_8520 = '%ID39'; Type_8520 = 'DINT'; AddressPointer_8520 = ADR(%ID39); AdrOffset_8530 = 4294967295; BitOffset_8530 = 0; BitLength_8530 = 0; Address_8530 = ''; Type_8530 = ''; AddressPointer_8530 = 0; AdrOffset_8540 = 4294967295;
              BitOffset_8540 = 0; BitLength_8540 = 0; Address_8540 = ''; Type_8540 = ''; AddressPointer_8540 = 0; AdrOffset_8550 = 152; BitOffset_8550 = 0; BitLength_8550 = 8; Address_8550 = '%IB152'; Type_8550 = 'SINT'; AddressPointer_8550 = ADR(%IB152); AdrOffset_8560 = 168; BitOffset_8560 = 0; BitLength_8560 = 32; Address_8560 = '%ID42'; Type_8560 = 'UDINT'; AddressPointer_8560 = ADR(%ID42); AdrOffset_8570 = 160; BitOffset_8570 = 0; BitLength_8570 = 16; Address_8570 = '%IW80'; Type_8570 = 'UINT'; AddressPointer_8570 = ADR(%IW80); AdrOffset_8580 = 164; BitOffset_8580 = 0; BitLength_8580 = 32; Address_8580 = '%ID41'; Type_8580 = 'DINT'; AddressPointer_8580 = ADR(%ID41); AdrOffset_8590 = 4294967295; BitOffset_8590 = 0; BitLength_8590 = 0; Address_8590 = ''; Type_8590 = ''; AddressPointer_8590 = 0; AdrOffset_8600 = 4294967295; BitOffset_8600 = 0; BitLength_8600 = 0; Address_8600 = ''; Type_8600 = '';
              AddressPointer_8600 = 0; AdrOffset_8600 = 4294967295; BitOffset_8600 = 0; BitLength_8600 = 0; Address_8610 = ''; Type_8610 = ''; AddressPointer_8610 = 0; AdrOffset_8620 = 4294967295; BitOffset_8620 = 0; BitLength_8620 = 0; Address_8620 = ''; Type_8620 = ''; AddressPointer_8620 = 0
    ModbusTCP_Slave_Device : Modbus TCP Slave, Leadshine Technology Co., Ltd., version 00.00.00.10
        settings: SlaveID = 1
*)

// Device/Application/PLC_PRG
PROGRAM PLC_PRG
VAR
	MC_Power_0: MC_Power;
	MC_Home_0: MC_Home;
	MC_Home_2: MC_Home;
	MC_Power_2: MC_Power;
	MC_Power_1: MC_Power;
	MC_Home_1: MC_Home;
	MC_Power_6: MC_Power;
	MC_Home_6: MC_Home;
	SMC_GroupPower_0: SMC_GroupPower;
	Status: BOOL;
	MC_GroupEnable_0: MC_GroupEnable;
	MC_SetCoordinateTransform_0: MC_SetCoordinateTransform;
	mcs: MC_COORD_REF;
	MC_HOME_3: MC_Home;
	MC_HOME_4: MC_Home;
	MC_HOME_5: MC_Home;
	MC_Reset_0: MC_Reset;
	MC_Reset_1: MC_Reset;
	MC_Reset_2: MC_Reset;
	MC_Reset_3: MC_Reset;
	MC_Reset_4: MC_Reset;
	MC_Reset_5: MC_Reset;
	MC_Reset_6: MC_Reset;
	mc_jog_for_biaoding: MC_Jog;
	MC_MoveDirectRelative_for_biaoding: MC_MoveDirectRelative;
	deltabd: SMC_POS_REF;
	ZJRED1: ARRAY [0..2] OF LREAL;
	ZJRED2: ARRAY [0..2] OF LREAL;
	ZJBLUE: ARRAY [0..2] OF LREAL;
	ZJYELLOW: ARRAY [0..2] OF LREAL;
	LS_3AxisLineAbs_zjzqred1: LS_3AxisLineAbs;
	zjzqred1: BOOL;
	LS_3AxisLineAbs_zjydred1: LS_3AxisLineAbs;
	POS1: ARRAY [0..2] OF LREAL;
	zjydred1: BOOL;
	LS_3AxisLineRel_zjfxred1: LS_3AxisLineRel;
	POS2: ARRAY [0..2] OF LREAL;
	zjfxred1: BOOL;
	LS_3AxisLineAbs_zjzqred2: LS_3AxisLineAbs;
	zjzqred2: BOOL;
	LS_3AxisLineAbs_zjydred2: LS_3AxisLineAbs;
	zjydred2: BOOL;
	LS_3AxisLineRel_zjfxred2: LS_3AxisLineRel;
	zjfxred2: BOOL;
	LS_3AxisLineAbs_zjzqblue: LS_3AxisLineAbs;
	zjzqblue: BOOL;
	LS_3AxisLineAbs_zjydblue: LS_3AxisLineAbs;
	zjydblue: BOOL;
	zjfxblue: BOOL;
	LS_3AxisLineRel_zjfxblue: LS_3AxisLineRel;
	MC_MoveAbsolute_0: MC_MoveAbsolute;
	dddelta: BOOL;
	MC_MoveDirectAbsolute_deltazqred: MC_MoveDirectAbsolute;
	deltazqredint: INT;
	deltazqred: BOOL;
	DELTAZQredpos: SMC_POS_REF;
	deltaykpos: SMC_POS_REF;
	zjfxbluem: BOOL;
	MC_MoveDirectAbsolute_deltayk: MC_MoveDirectAbsolute;
	zjpz: INT;
	deltapz: INT;
	deltaqzred: BOOL;
	MC_MoveDirectAbsolute_deltaydred: MC_MoveDirectAbsolute;
	MC_Halt_0: MC_Halt;
	MC_Halt_1: MC_Halt;
	MC_Halt_2: MC_Halt;
	MC_Halt_3: MC_Halt;
	MC_Halt_4: MC_Halt;
	MC_Halt_5: MC_Halt;
	MC_Halt_6: MC_Halt;
	DELTAYDredpos: SMC_POS_REF;
	deltaydred: BOOL;
	MC_MoveDirectRelative_deltafxred: MC_MoveDirectRelative;
	DELTAYD2FX: SMC_POS_REF;
	deltazqblue: BOOL;
	deltafxred: BOOL;
	deltafxblue: BOOL;
	deltaqyk: BOOL;
	deltayk: BOOL;
	deltafxbluem: BOOL;
	deltafxredm: BOOL;
	TON_0: TON;
	deltafxred1: BOOL;
	deltazqblueint: INT;
	deltaqzblue: BOOL;
	MC_MoveDirectAbsolute_deltazqblue: MC_MoveDirectAbsolute;
	DELTAZQbluepos: SMC_POS_REF;
	MC_MoveDirectAbsolute_deltaydblue: MC_MoveDirectAbsolute;
	DELTAYDbluepos: SMC_POS_REF;
	deltaydblue: BOOL;
	MC_MoveDirectRelative_deltafxblue: MC_MoveDirectRelative;
	deltafxblue1: BOOL;
	TON_1: TON;
END_VAR
VAR // added by the converter: edge detectors and wires of the graphical bodies
    _rt1, _rt2, _rt3, _rt4, _rt5, _rt6, _rt7, _rt8, _rt9, _rt10, _rt11, _rt12, _rt13, _rt14, _rt15 : R_TRIG;
END_VAR

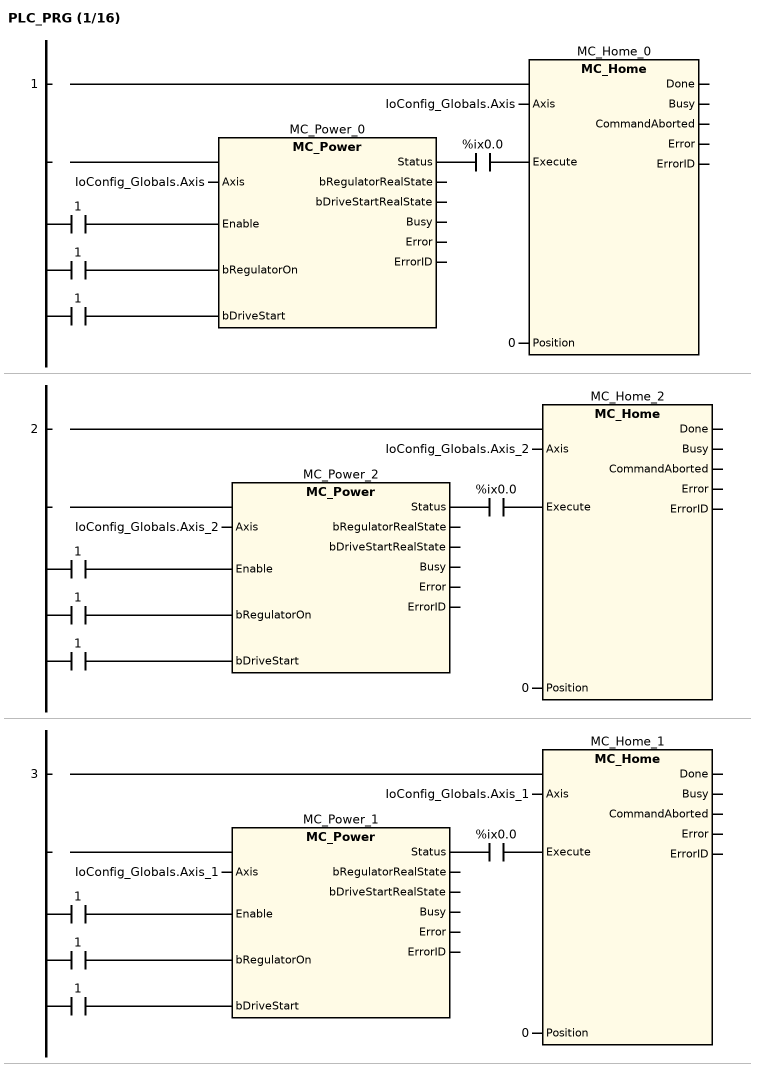
// NETWORK 1
MC_Power_0(Axis := IoConfig_Globals.Axis, Enable := 1, bRegulatorOn := 1, bDriveStart := 1); // MC_Power
MC_Home_0(Axis := IoConfig_Globals.Axis, Execute := MC_Power_0.Status AND %ix0.0, Position := 0); // MC_Home

// NETWORK 2
MC_Power_2(Axis := IoConfig_Globals.Axis_2, Enable := 1, bRegulatorOn := 1, bDriveStart := 1); // MC_Power
MC_Home_2(Axis := IoConfig_Globals.Axis_2, Execute := MC_Power_2.Status AND %ix0.0, Position := 0); // MC_Home

// NETWORK 3
MC_Power_1(Axis := IoConfig_Globals.Axis_1, Enable := 1, bRegulatorOn := 1, bDriveStart := 1); // MC_Power
MC_Home_1(Axis := IoConfig_Globals.Axis_1, Execute := MC_Power_1.Status AND %ix0.0, Position := 0); // MC_Home

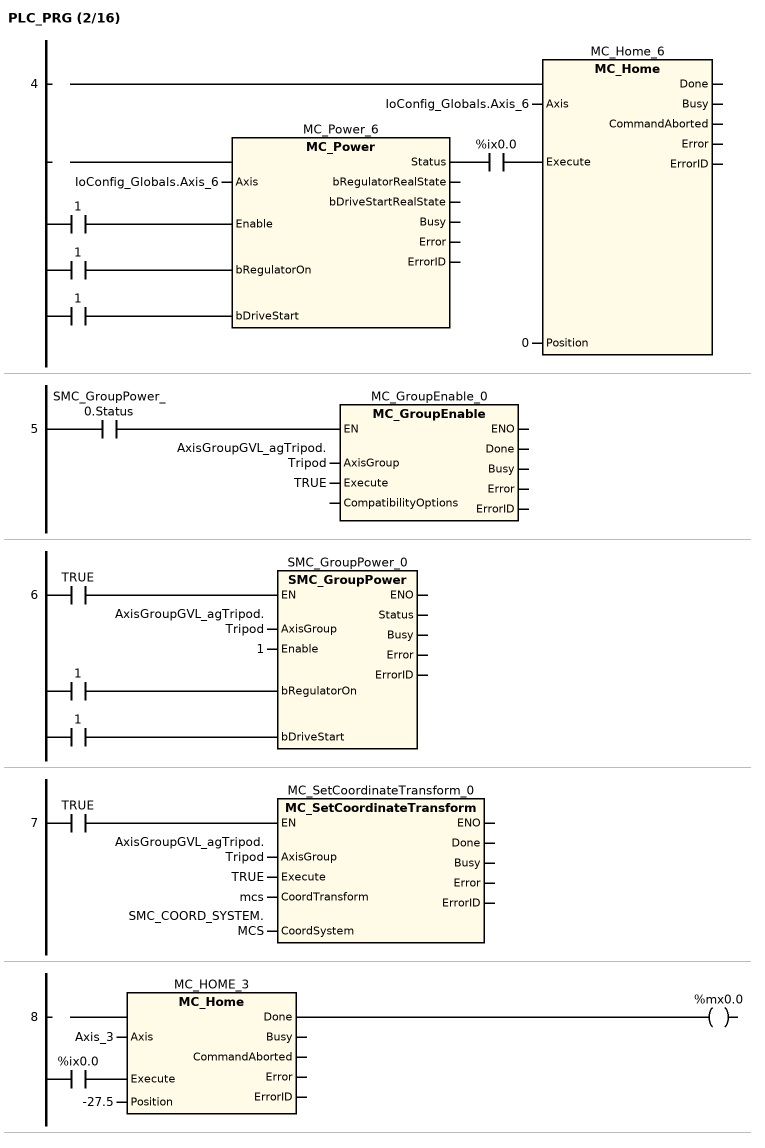
// NETWORK 4
MC_Power_6(Axis := IoConfig_Globals.Axis_6, Enable := 1, bRegulatorOn := 1, bDriveStart := 1); // MC_Power
MC_Home_6(Axis := IoConfig_Globals.Axis_6, Execute := MC_Power_6.Status AND %ix0.0, Position := 0); // MC_Home

// NETWORK 5
IF SMC_GroupPower_0.Status THEN
    MC_GroupEnable_0(AxisGroup := AxisGroupGVL_agTripod.Tripod, Execute := TRUE); // MC_GroupEnable
END_IF

// NETWORK 6
SMC_GroupPower_0(AxisGroup := AxisGroupGVL_agTripod.Tripod, Enable := 1, bRegulatorOn := 1, bDriveStart := 1); // SMC_GroupPower

// NETWORK 7
MC_SetCoordinateTransform_0(
    AxisGroup := AxisGroupGVL_agTripod.Tripod,
    Execute := TRUE,
    CoordTransform := mcs,
    CoordSystem := SMC_COORD_SYSTEM.MCS); // MC_SetCoordinateTransform

// NETWORK 8
MC_HOME_3(Axis := Axis_3, Execute := %ix0.0, Position := -27.5); // MC_Home
%mx0.0 := MC_HOME_3.Done;

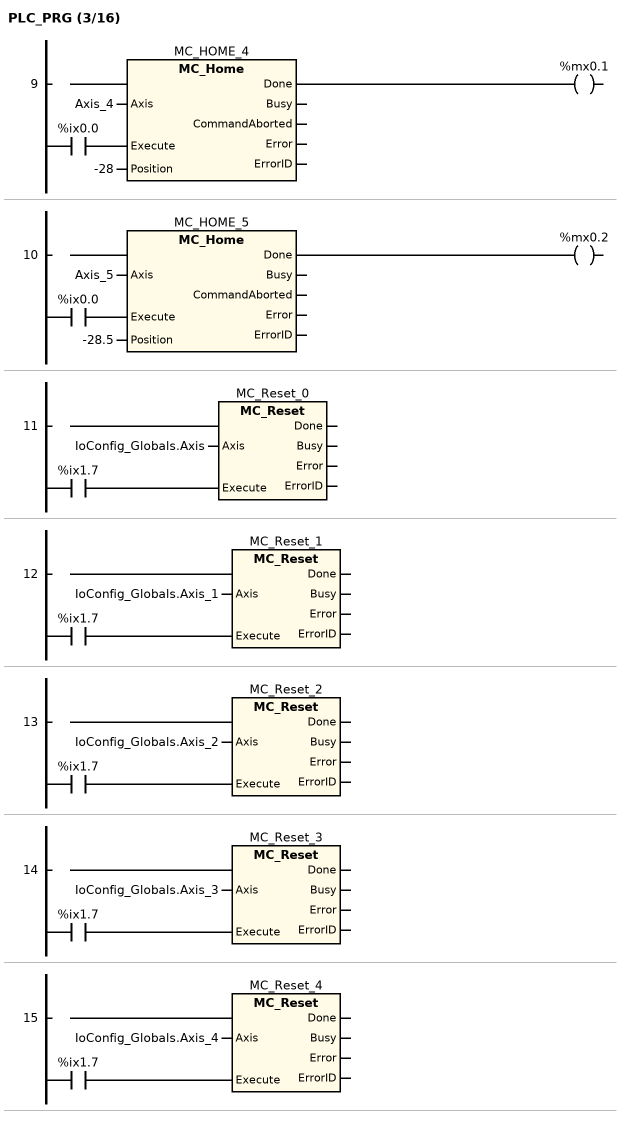
// NETWORK 9
MC_HOME_4(Axis := Axis_4, Execute := %ix0.0, Position := -28); // MC_Home
%mx0.1 := MC_HOME_4.Done;

// NETWORK 10
MC_HOME_5(Axis := Axis_5, Execute := %ix0.0, Position := -28.5); // MC_Home
%mx0.2 := MC_HOME_5.Done;

// NETWORK 11
MC_Reset_0(Axis := IoConfig_Globals.Axis, Execute := %ix1.7); // MC_Reset

// NETWORK 12
MC_Reset_1(Axis := IoConfig_Globals.Axis_1, Execute := %ix1.7); // MC_Reset

// NETWORK 13
MC_Reset_2(Axis := IoConfig_Globals.Axis_2, Execute := %ix1.7); // MC_Reset

// NETWORK 14
MC_Reset_3(Axis := IoConfig_Globals.Axis_3, Execute := %ix1.7); // MC_Reset

// NETWORK 15
MC_Reset_4(Axis := IoConfig_Globals.Axis_4, Execute := %ix1.7); // MC_Reset

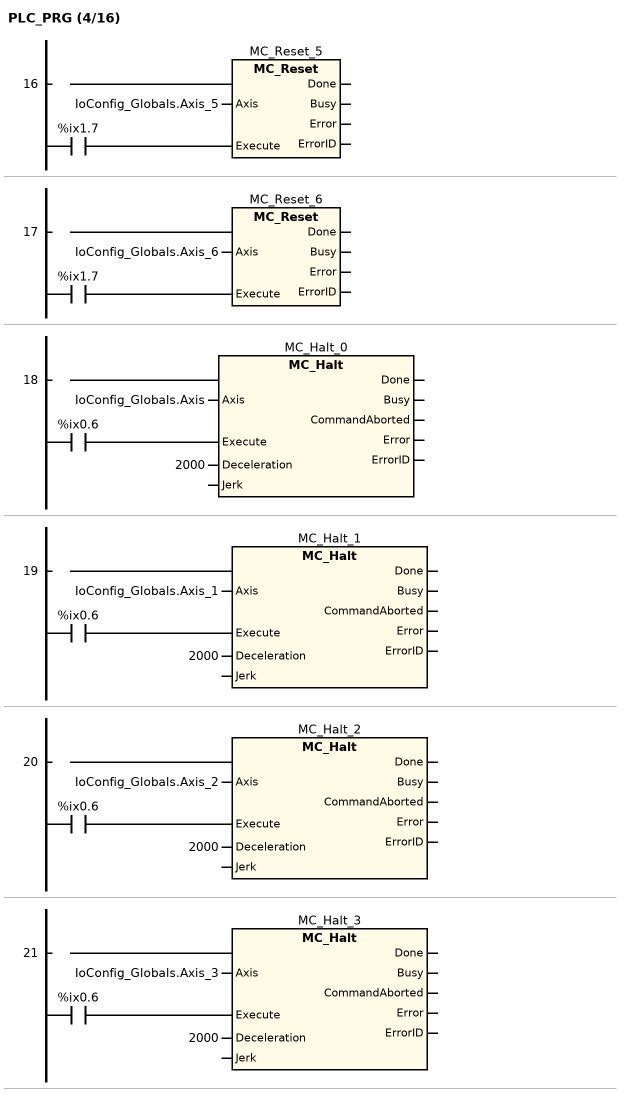
// NETWORK 16
MC_Reset_5(Axis := IoConfig_Globals.Axis_5, Execute := %ix1.7); // MC_Reset

// NETWORK 17
MC_Reset_6(Axis := IoConfig_Globals.Axis_6, Execute := %ix1.7); // MC_Reset

// NETWORK 18
MC_Halt_0(Axis := IoConfig_Globals.Axis, Execute := %ix0.6, Deceleration := 2000); // MC_Halt

// NETWORK 19
MC_Halt_1(Axis := IoConfig_Globals.Axis_1, Execute := %ix0.6, Deceleration := 2000); // MC_Halt

// NETWORK 20
MC_Halt_2(Axis := IoConfig_Globals.Axis_2, Execute := %ix0.6, Deceleration := 2000); // MC_Halt

// NETWORK 21
MC_Halt_3(Axis := IoConfig_Globals.Axis_3, Execute := %ix0.6, Deceleration := 2000); // MC_Halt

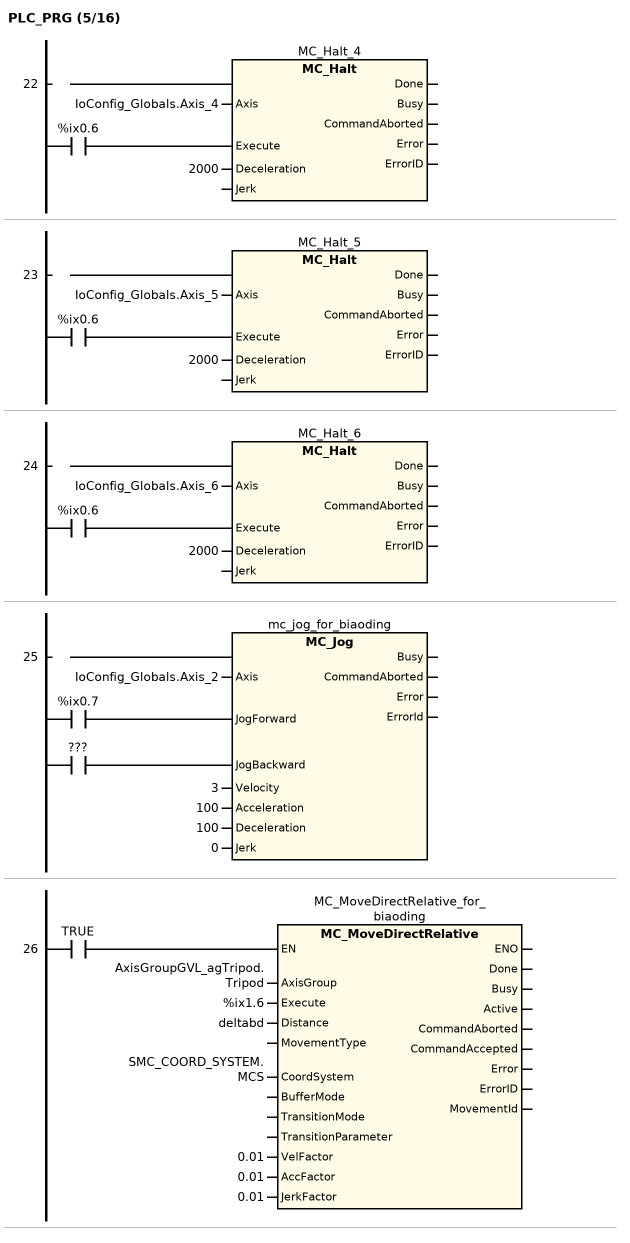
// NETWORK 22
MC_Halt_4(Axis := IoConfig_Globals.Axis_4, Execute := %ix0.6, Deceleration := 2000); // MC_Halt

// NETWORK 23
MC_Halt_5(Axis := IoConfig_Globals.Axis_5, Execute := %ix0.6, Deceleration := 2000); // MC_Halt

// NETWORK 24
MC_Halt_6(Axis := IoConfig_Globals.Axis_6, Execute := %ix0.6, Deceleration := 2000); // MC_Halt

// NETWORK 25
mc_jog_for_biaoding(
    Axis := IoConfig_Globals.Axis_2,
    JogForward := %ix0.7,
    Velocity := 3,
    Acceleration := 100,
    Deceleration := 100,
    Jerk := 0); // MC_Jog

// NETWORK 26
MC_MoveDirectRelative_for_biaoding(
    AxisGroup := AxisGroupGVL_agTripod.Tripod,
    Execute := %ix1.6,
    Distance := deltabd,
    CoordSystem := SMC_COORD_SYSTEM.MCS,
    VelFactor := 0.01,
    AccFactor := 0.01,
    JerkFactor := 0.01); // MC_MoveDirectRelative

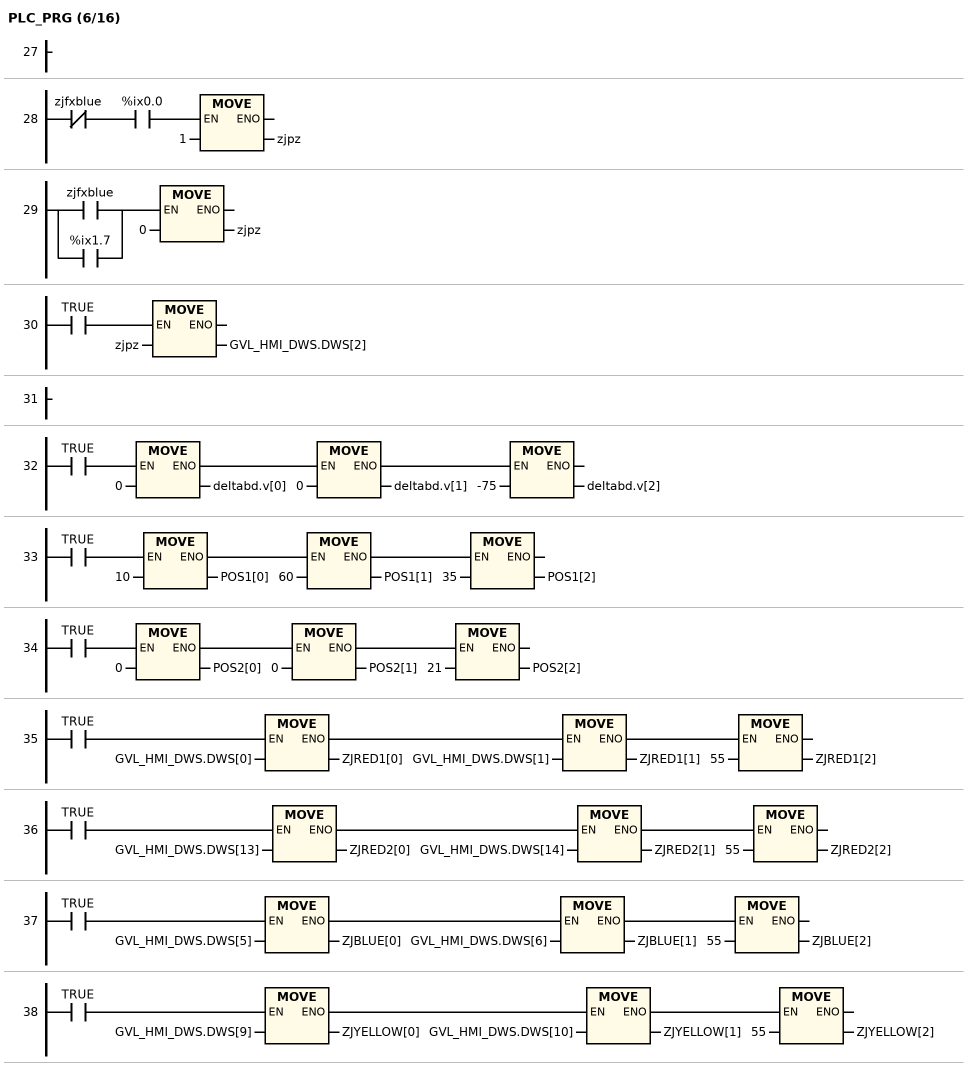
// NETWORK 27

// NETWORK 28
IF NOT zjfxblue AND %ix0.0 THEN zjpz := 1; END_IF

// NETWORK 29
IF zjfxblue OR %ix1.7 THEN zjpz := 0; END_IF

// NETWORK 30
GVL_HMI_DWS.DWS[2] := zjpz;

// NETWORK 31

// NETWORK 32
deltabd.v[0] := 0;
deltabd.v[1] := 0;
deltabd.v[2] := -75;

// NETWORK 33
POS1[0] := 10;
POS1[1] := 60;
POS1[2] := 35;

// NETWORK 34
POS2[0] := 0;
POS2[1] := 0;
POS2[2] := 21;

// NETWORK 35
ZJRED1[0] := GVL_HMI_DWS.DWS[0];
ZJRED1[1] := GVL_HMI_DWS.DWS[1];
ZJRED1[2] := 55;

// NETWORK 36
ZJRED2[0] := GVL_HMI_DWS.DWS[13];
ZJRED2[1] := GVL_HMI_DWS.DWS[14];
ZJRED2[2] := 55;

// NETWORK 37
ZJBLUE[0] := GVL_HMI_DWS.DWS[5];
ZJBLUE[1] := GVL_HMI_DWS.DWS[6];
ZJBLUE[2] := 55;

// NETWORK 38
ZJYELLOW[0] := GVL_HMI_DWS.DWS[9];
ZJYELLOW[1] := GVL_HMI_DWS.DWS[10];
ZJYELLOW[2] := 55;

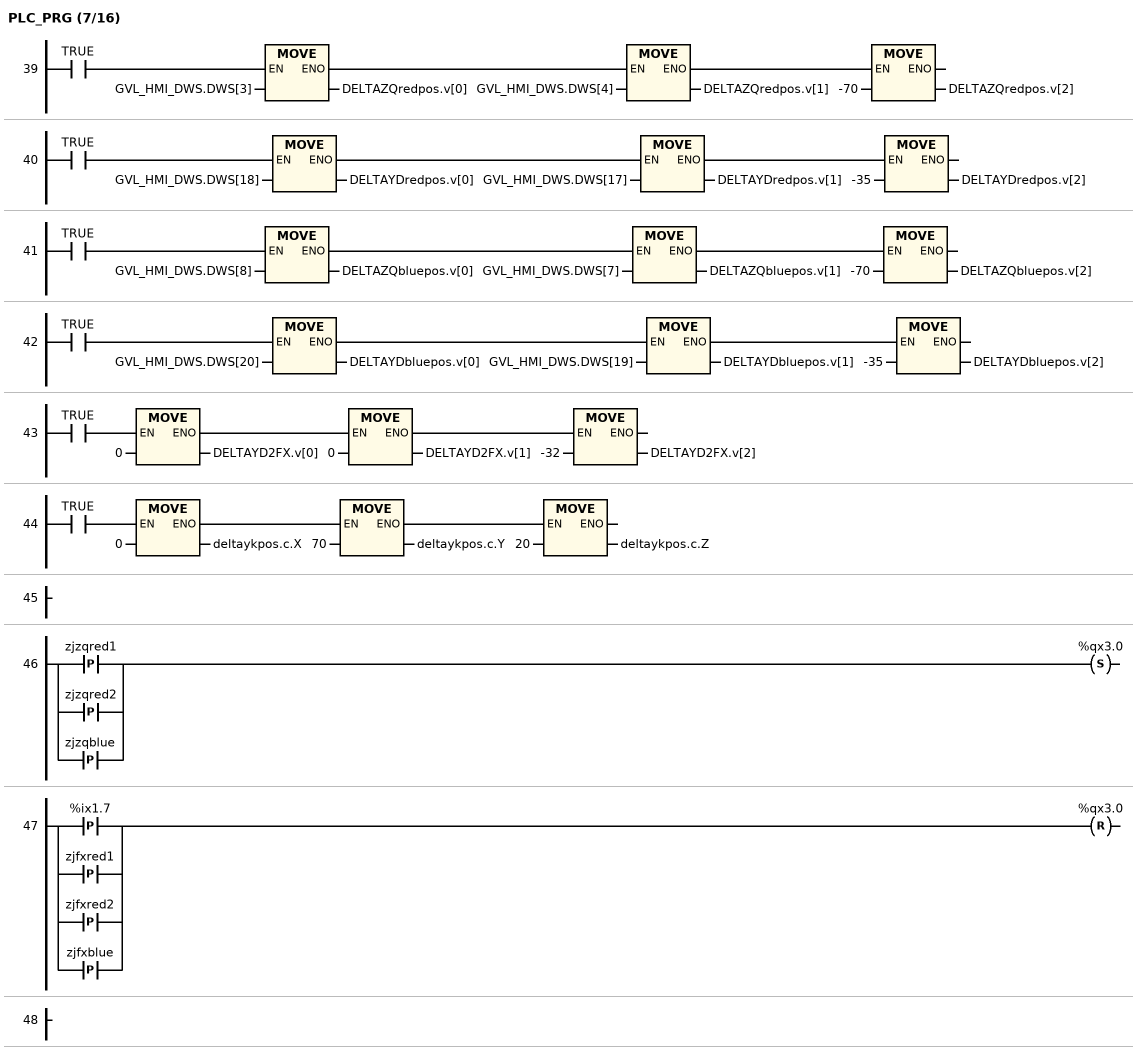
// NETWORK 39
DELTAZQredpos.v[0] := GVL_HMI_DWS.DWS[3];
DELTAZQredpos.v[1] := GVL_HMI_DWS.DWS[4];
DELTAZQredpos.v[2] := -70;

// NETWORK 40
DELTAYDredpos.v[0] := GVL_HMI_DWS.DWS[18];
DELTAYDredpos.v[1] := GVL_HMI_DWS.DWS[17];
DELTAYDredpos.v[2] := -35;

// NETWORK 41
DELTAZQbluepos.v[0] := GVL_HMI_DWS.DWS[8];
DELTAZQbluepos.v[1] := GVL_HMI_DWS.DWS[7];
DELTAZQbluepos.v[2] := -70;

// NETWORK 42
DELTAYDbluepos.v[0] := GVL_HMI_DWS.DWS[20];
DELTAYDbluepos.v[1] := GVL_HMI_DWS.DWS[19];
DELTAYDbluepos.v[2] := -35;

// NETWORK 43
DELTAYD2FX.v[0] := 0;
DELTAYD2FX.v[1] := 0;
DELTAYD2FX.v[2] := -32;

// NETWORK 44
deltaykpos.c.X := 0;
deltaykpos.c.Y := 70;
deltaykpos.c.Z := 20;

// NETWORK 45

// NETWORK 46
_rt1(CLK := zjzqred1);
_rt2(CLK := zjzqred2);
_rt3(CLK := zjzqblue);
%qx3.0 S= _rt1.Q OR _rt2.Q OR _rt3.Q;

// NETWORK 47
_rt4(CLK := %ix1.7);
_rt5(CLK := zjfxred1);
_rt6(CLK := zjfxred2);
_rt7(CLK := zjfxblue);
%qx3.0 R= _rt4.Q OR _rt5.Q OR _rt6.Q OR _rt7.Q;

// NETWORK 48

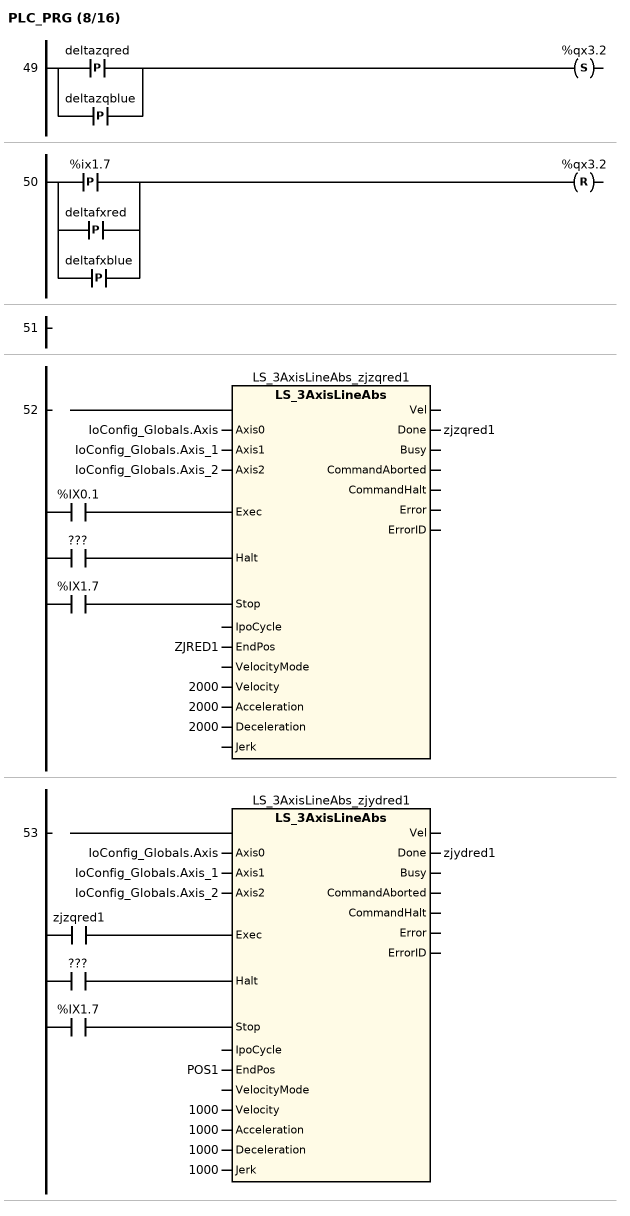
// NETWORK 49
_rt8(CLK := deltazqred);
_rt9(CLK := deltazqblue);
%qx3.2 S= _rt8.Q OR _rt9.Q;

// NETWORK 50
_rt10(CLK := %ix1.7);
_rt11(CLK := deltafxred);
_rt12(CLK := deltafxblue);
%qx3.2 R= _rt10.Q OR _rt11.Q OR _rt12.Q;

// NETWORK 51

// NETWORK 52
LS_3AxisLineAbs_zjzqred1(
    Axis0 := IoConfig_Globals.Axis,
    Axis1 := IoConfig_Globals.Axis_1,
    Axis2 := IoConfig_Globals.Axis_2,
    Exec := %IX0.1,
    Stop := %IX1.7,
    EndPos := ZJRED1,
    Velocity := 2000,
    Acceleration := 2000,
    Deceleration := 2000,
    Done => zjzqred1); // LS_3AxisLineAbs

// NETWORK 53
LS_3AxisLineAbs_zjydred1(
    Axis0 := IoConfig_Globals.Axis,
    Axis1 := IoConfig_Globals.Axis_1,
    Axis2 := IoConfig_Globals.Axis_2,
    Exec := zjzqred1,
    Stop := %IX1.7,
    EndPos := POS1,
    Velocity := 1000,
    Acceleration := 1000,
    Deceleration := 1000,
    Jerk := 1000,
    Done => zjydred1); // LS_3AxisLineAbs

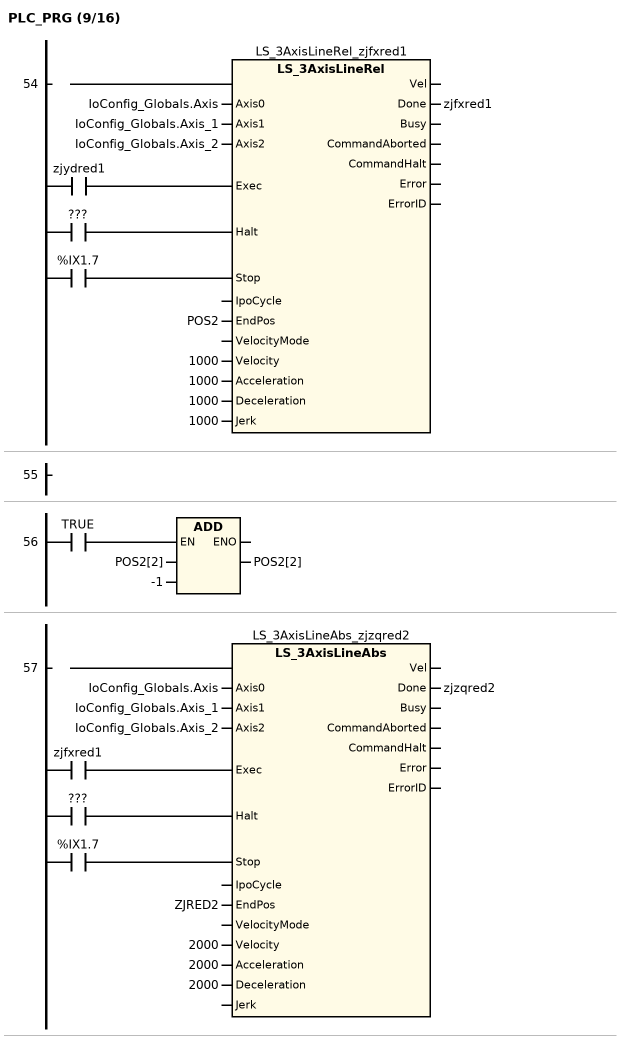
// NETWORK 54
LS_3AxisLineRel_zjfxred1(
    Axis0 := IoConfig_Globals.Axis,
    Axis1 := IoConfig_Globals.Axis_1,
    Axis2 := IoConfig_Globals.Axis_2,
    Exec := zjydred1,
    Stop := %IX1.7,
    EndPos := POS2,
    Velocity := 1000,
    Acceleration := 1000,
    Deceleration := 1000,
    Jerk := 1000,
    Done => zjfxred1); // LS_3AxisLineRel

// NETWORK 55

// NETWORK 56
POS2[2] := POS2[2] + -1;

// NETWORK 57
LS_3AxisLineAbs_zjzqred2(
    Axis0 := IoConfig_Globals.Axis,
    Axis1 := IoConfig_Globals.Axis_1,
    Axis2 := IoConfig_Globals.Axis_2,
    Exec := zjfxred1,
    Stop := %IX1.7,
    EndPos := ZJRED2,
    Velocity := 2000,
    Acceleration := 2000,
    Deceleration := 2000,
    Done => zjzqred2); // LS_3AxisLineAbs

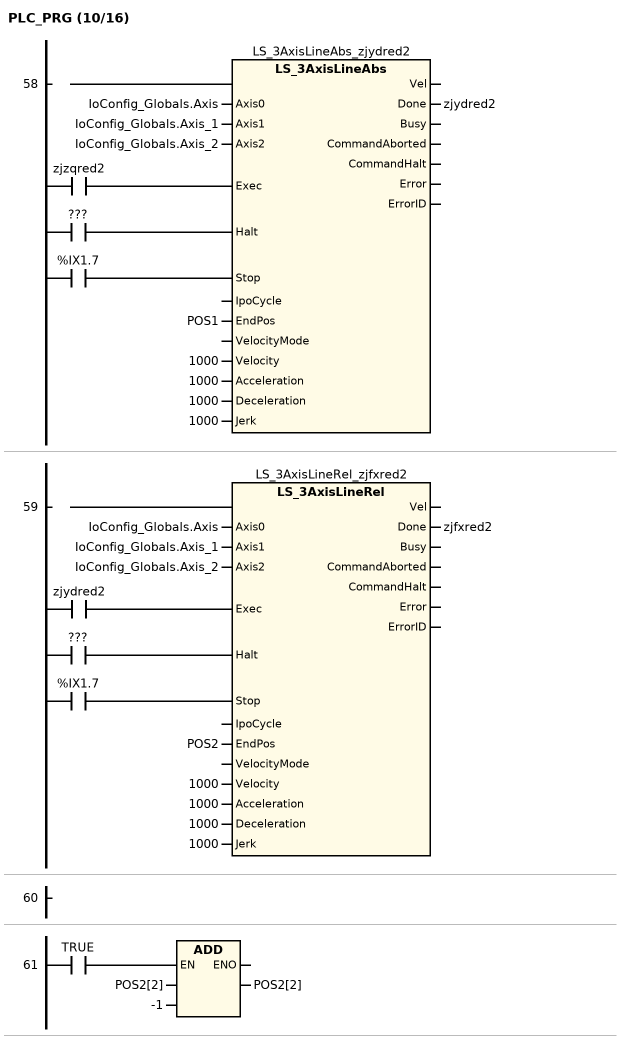
// NETWORK 58
LS_3AxisLineAbs_zjydred2(
    Axis0 := IoConfig_Globals.Axis,
    Axis1 := IoConfig_Globals.Axis_1,
    Axis2 := IoConfig_Globals.Axis_2,
    Exec := zjzqred2,
    Stop := %IX1.7,
    EndPos := POS1,
    Velocity := 1000,
    Acceleration := 1000,
    Deceleration := 1000,
    Jerk := 1000,
    Done => zjydred2); // LS_3AxisLineAbs

// NETWORK 59
LS_3AxisLineRel_zjfxred2(
    Axis0 := IoConfig_Globals.Axis,
    Axis1 := IoConfig_Globals.Axis_1,
    Axis2 := IoConfig_Globals.Axis_2,
    Exec := zjydred2,
    Stop := %IX1.7,
    EndPos := POS2,
    Velocity := 1000,
    Acceleration := 1000,
    Deceleration := 1000,
    Jerk := 1000,
    Done => zjfxred2); // LS_3AxisLineRel

// NETWORK 60

// NETWORK 61
POS2[2] := POS2[2] + -1;

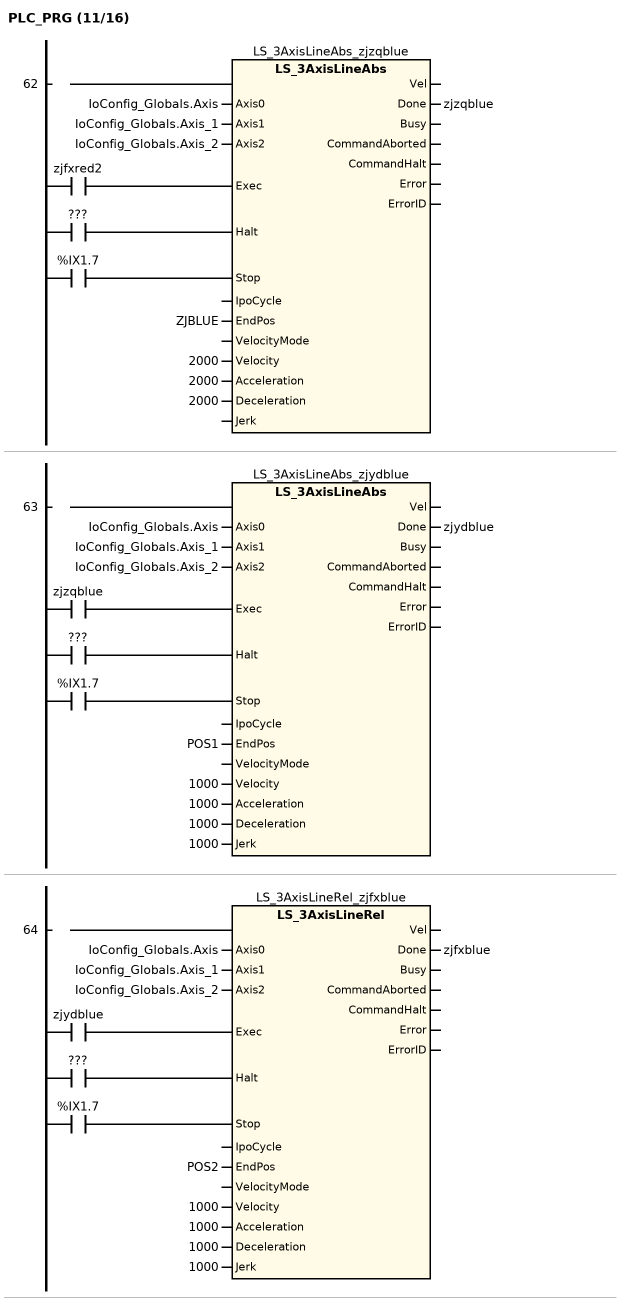
// NETWORK 62
LS_3AxisLineAbs_zjzqblue(
    Axis0 := IoConfig_Globals.Axis,
    Axis1 := IoConfig_Globals.Axis_1,
    Axis2 := IoConfig_Globals.Axis_2,
    Exec := zjfxred2,
    Stop := %IX1.7,
    EndPos := ZJBLUE,
    Velocity := 2000,
    Acceleration := 2000,
    Deceleration := 2000,
    Done => zjzqblue); // LS_3AxisLineAbs

// NETWORK 63
LS_3AxisLineAbs_zjydblue(
    Axis0 := IoConfig_Globals.Axis,
    Axis1 := IoConfig_Globals.Axis_1,
    Axis2 := IoConfig_Globals.Axis_2,
    Exec := zjzqblue,
    Stop := %IX1.7,
    EndPos := POS1,
    Velocity := 1000,
    Acceleration := 1000,
    Deceleration := 1000,
    Jerk := 1000,
    Done => zjydblue); // LS_3AxisLineAbs

// NETWORK 64
LS_3AxisLineRel_zjfxblue(
    Axis0 := IoConfig_Globals.Axis,
    Axis1 := IoConfig_Globals.Axis_1,
    Axis2 := IoConfig_Globals.Axis_2,
    Exec := zjydblue,
    Stop := %IX1.7,
    EndPos := POS2,
    Velocity := 1000,
    Acceleration := 1000,
    Deceleration := 1000,
    Jerk := 1000,
    Done => zjfxblue); // LS_3AxisLineRel

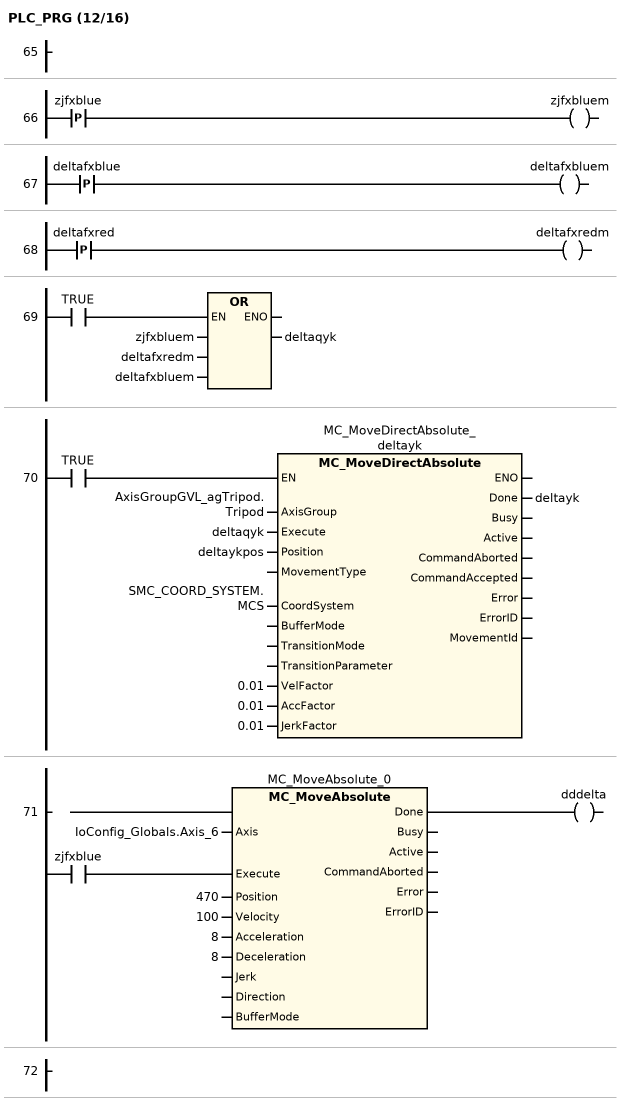
// NETWORK 65

// NETWORK 66
_rt13(CLK := zjfxblue);
zjfxbluem := _rt13.Q;

// NETWORK 67
_rt14(CLK := deltafxblue);
deltafxbluem := _rt14.Q;

// NETWORK 68
_rt15(CLK := deltafxred);
deltafxredm := _rt15.Q;

// NETWORK 69
deltaqyk := zjfxbluem OR deltafxredm OR deltafxbluem;

// NETWORK 70
MC_MoveDirectAbsolute_deltayk(
    AxisGroup := AxisGroupGVL_agTripod.Tripod,
    Execute := deltaqyk,
    Position := deltaykpos,
    CoordSystem := SMC_COORD_SYSTEM.MCS,
    VelFactor := 0.01,
    AccFactor := 0.01,
    JerkFactor := 0.01,
    Done => deltayk); // MC_MoveDirectAbsolute

// NETWORK 71
MC_MoveAbsolute_0(
    Axis := IoConfig_Globals.Axis_6,
    Execute := zjfxblue,
    Position := 470,
    Velocity := 100,
    Acceleration := 8,
    Deceleration := 8); // MC_MoveAbsolute
dddelta := MC_MoveAbsolute_0.Done;

// NETWORK 72

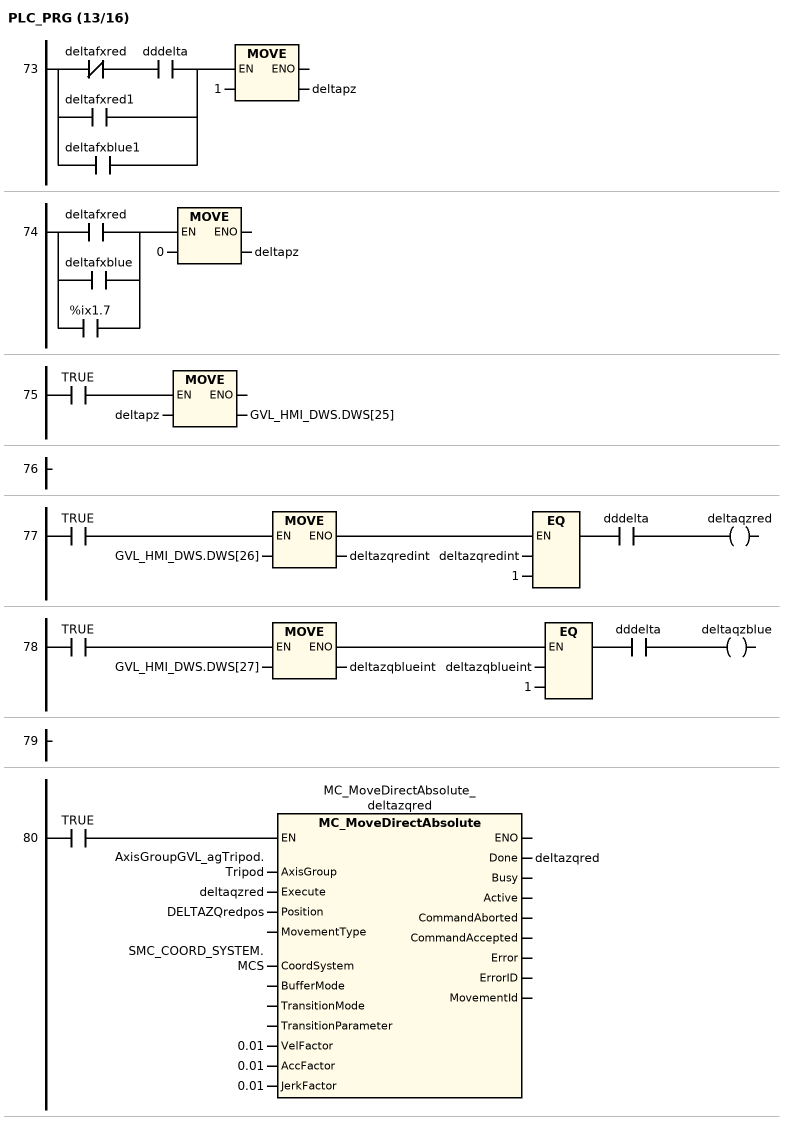
// NETWORK 73
IF NOT deltafxred AND dddelta OR deltafxred1 OR deltafxblue1 THEN deltapz := 1; END_IF

// NETWORK 74
IF deltafxred OR deltafxblue OR %ix1.7 THEN deltapz := 0; END_IF

// NETWORK 75
GVL_HMI_DWS.DWS[25] := deltapz;

// NETWORK 76

// NETWORK 77
deltazqredint := GVL_HMI_DWS.DWS[26];
deltaqzred := deltazqredint = 1 AND dddelta;

// NETWORK 78
deltazqblueint := GVL_HMI_DWS.DWS[27];
deltaqzblue := deltazqblueint = 1 AND dddelta;

// NETWORK 79

// NETWORK 80
MC_MoveDirectAbsolute_deltazqred(
    AxisGroup := AxisGroupGVL_agTripod.Tripod,
    Execute := deltaqzred,
    Position := DELTAZQredpos,
    CoordSystem := SMC_COORD_SYSTEM.MCS,
    VelFactor := 0.01,
    AccFactor := 0.01,
    JerkFactor := 0.01,
    Done => deltazqred); // MC_MoveDirectAbsolute

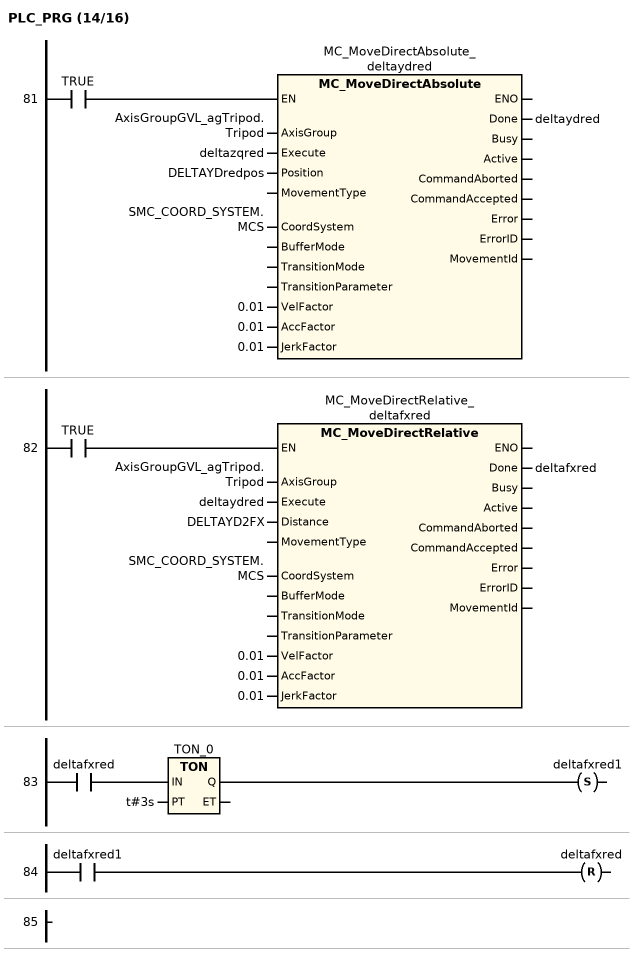
// NETWORK 81
MC_MoveDirectAbsolute_deltaydred(
    AxisGroup := AxisGroupGVL_agTripod.Tripod,
    Execute := deltazqred,
    Position := DELTAYDredpos,
    CoordSystem := SMC_COORD_SYSTEM.MCS,
    VelFactor := 0.01,
    AccFactor := 0.01,
    JerkFactor := 0.01,
    Done => deltaydred); // MC_MoveDirectAbsolute

// NETWORK 82
MC_MoveDirectRelative_deltafxred(
    AxisGroup := AxisGroupGVL_agTripod.Tripod,
    Execute := deltaydred,
    Distance := DELTAYD2FX,
    CoordSystem := SMC_COORD_SYSTEM.MCS,
    VelFactor := 0.01,
    AccFactor := 0.01,
    JerkFactor := 0.01,
    Done => deltafxred); // MC_MoveDirectRelative

// NETWORK 83
TON_0(IN := deltafxred, PT := t#3s); // TON
deltafxred1 S= TON_0.Q;

// NETWORK 84
deltafxred R= deltafxred1;

// NETWORK 85

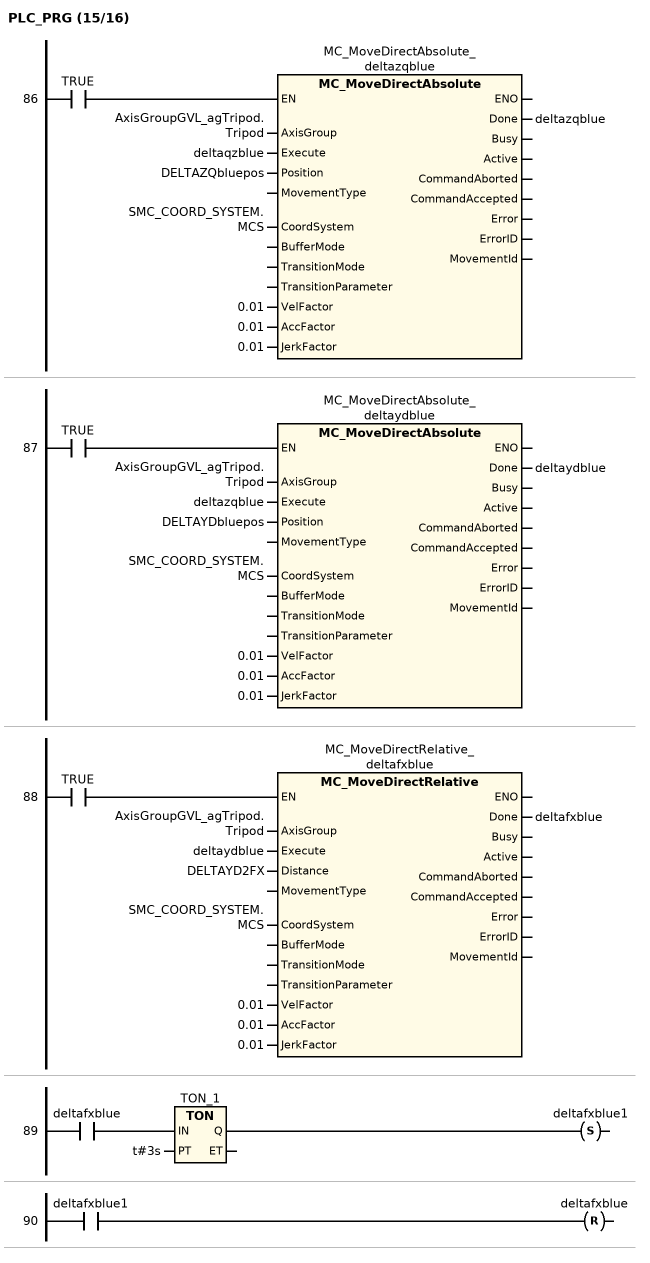
// NETWORK 86
MC_MoveDirectAbsolute_deltazqblue(
    AxisGroup := AxisGroupGVL_agTripod.Tripod,
    Execute := deltaqzblue,
    Position := DELTAZQbluepos,
    CoordSystem := SMC_COORD_SYSTEM.MCS,
    VelFactor := 0.01,
    AccFactor := 0.01,
    JerkFactor := 0.01,
    Done => deltazqblue); // MC_MoveDirectAbsolute

// NETWORK 87
MC_MoveDirectAbsolute_deltaydblue(
    AxisGroup := AxisGroupGVL_agTripod.Tripod,
    Execute := deltazqblue,
    Position := DELTAYDbluepos,
    CoordSystem := SMC_COORD_SYSTEM.MCS,
    VelFactor := 0.01,
    AccFactor := 0.01,
    JerkFactor := 0.01,
    Done => deltaydblue); // MC_MoveDirectAbsolute

// NETWORK 88
MC_MoveDirectRelative_deltafxblue(
    AxisGroup := AxisGroupGVL_agTripod.Tripod,
    Execute := deltaydblue,
    Distance := DELTAYD2FX,
    CoordSystem := SMC_COORD_SYSTEM.MCS,
    VelFactor := 0.01,
    AccFactor := 0.01,
    JerkFactor := 0.01,
    Done => deltafxblue); // MC_MoveDirectRelative

// NETWORK 89
TON_1(IN := deltafxblue, PT := t#3s); // TON
deltafxblue1 S= TON_1.Q;

// NETWORK 90
deltafxblue R= deltafxblue1;

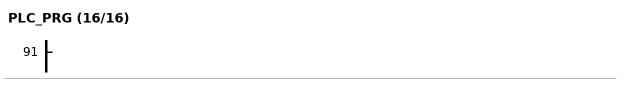
// NETWORK 91

END_PROGRAM
